LIN {X 0,Y 516.886,Z 290.1,A -85,B 0,C 180,E1 -5001.285,E2 -5001.285} C_VEL
LIN {X 0,Y 516.874,Z 290.104,A -85,B 0,C 180,E1 -5004.22,E2 -5004.22} C_VEL
LIN {X 0,Y 516.884,Z 290.103,A -85,B 0,C 180,E1 -5007.052,E2 -5007.052} C_VEL
LIN {X 0,Y 516.896,Z 290.1,A -85,B 0,C 180,E1 -5009.797,E2 -5009.797} C_VEL
LIN {X 0,Y 516.926,Z 290.096,A -85,B 0,C 180,E1 -5012.467,E2 -5012.467} C_VEL
LIN {X 0,Y 516.86,Z 290.106,A -85,B 0,C 180,E1 -5015.069,E2 -5015.069} C_VEL
LIN {X 0,Y 516.873,Z 290.103,A -85,B 0,C 180,E1 -5017.622,E2 -5017.622} C_VEL
LIN {X 0,Y 516.936,Z 290.095,A -85,B 0,C 180,E1 -5020.13,E2 -5020.13} C_VEL
LIN {X 0,Y 516.909,Z 290.098,A -85,B 0,C 180,E1 -5022.596,E2 -5022.596} C_VEL
LIN {X 0,Y 516.948,Z 290.093,A -85,B 0,C 180,E1 -5025.03,E2 -5025.03} C_VEL
LIN {X 0,Y 516.971,Z 290.091,A -85,B 0,C 180,E1 -5028.234,E2 -5028.234} C_VEL
LIN {X 0,Y 516.96,Z 290.091,A -85,B 0,C 180,E1 -5031.4,E2 -5031.4} C_VEL
LIN {X 0,Y 517.015,Z 290.083,A -85,B 0,C 180,E1 -5033.757,E2 -5033.757} C_VEL
LIN {X 0,Y 517.088,Z 290.074,A -85,B 0,C 180,E1 -5037.663,E2 -5037.663} C_VEL
LIN {X 0,Y 517.097,Z 290.075,A -85,B 0,C 180,E1 -5040.779,E2 -5040.779} C_VEL
LIN {X 0,Y 516.98,Z 290.089,A -85,B 0,C 180,E1 -5043.117,E2 -5043.117} C_VEL
LIN {X 0,Y 516.994,Z 290.088,A -85,B 0,C 180,E1 -5046.243,E2 -5046.243} C_VEL
LIN {X 0,Y 516.948,Z 290.092,A -85,B 0,C 180,E1 -5049.389,E2 -5049.389} C_VEL
LIN {X 0,Y 516.957,Z 290.093,A -85,B 0,C 180,E1 -5051.807,E2 -5051.807} C_VEL
LIN {X 0,Y 516.945,Z 290.093,A -85,B 0,C 180,E1 -5055.144,E2 -5055.144} C_VEL
LIN {X 0,Y 516.918,Z 290.099,A -85,B 0,C 180,E1 -5058.223,E2 -5058.223} C_VEL
LIN {X 0,Y 516.917,Z 290.099,A -85,B 0,C 180,E1 -5060.701,E2 -5060.701} C_VEL
LIN {X 0,Y 516.894,Z 290.099,A -85,B 0,C 180,E1 -5064.073,E2 -5064.073} C_VEL
LIN {X 0,Y 516.895,Z 290.099,A -85,B 0,C 180,E1 -5066.66,E2 -5066.66} C_VEL
LIN {X 0,Y 516.913,Z 290.096,A -85,B 0,C 180,E1 -5069.523,E2 -5069.523} C_VEL
LIN {X 0,Y 516.9,Z 290.102,A -85,B 0,C 180,E1 -5072.543,E2 -5072.543} C_VEL
LIN {X 0,Y 516.867,Z 290.104,A -85,B 0,C 180,E1 -5075.329,E2 -5075.329} C_VEL
LIN {X 0,Y 516.883,Z 290.104,A -85,B 0,C 180,E1 -5077.943,E2 -5077.943} C_VEL
LIN {X 0,Y 516.886,Z 290.101,A -85,B 0,C 180,E1 -5080.742,E2 -5080.742} C_VEL
LIN {X 0,Y 516.885,Z 290.101,A -85,B 0,C 180,E1 -5083.903,E2 -5083.903} C_VEL
LIN {X 0,Y 516.885,Z 290.1,A -85,B 0,C 180,E1 -5086.107,E2 -5086.107} C_VEL
LIN {X 0,Y 516.885,Z 290.1,A -85,B 0,C 180,E1 -5089.258,E2 -5089.258} C_VEL
LIN {X 0,Y 516.916,Z 290.213,A -85,B 0,C 180,E1 -5091.487,E2 -5091.487} C_VEL
LIN {X 0,Y 518.112,Z 296.915,A -85,B 0,C 180,E1 -5093.838,E2 -5093.838} C_VEL
LIN {X 0,Y 518.102,Z 303.042,A -85,B 0,C 180,E1 -5095.839,E2 -5095.839} C_VEL
LIN {X 0,Y 517.763,Z 312.405,A -85,B 0,C 180,E1 -5098.776,E2 -5098.776} C_VEL
LIN {X 0,Y 517.485,Z 322.995,A -85,B 0,C 180,E1 -5101.979,E2 -5101.979} C_VEL
LIN {X 0,Y 517.191,Z 333.621,A -85,B 0,C 180,E1 -5105.086,E2 -5105.086} C_VEL
LIN {X 0,Y 516.956,Z 344.077,A -85,B 0,C 180,E1 -5108.046,E2 -5108.046} C_VEL
LIN {X 0,Y 516.804,Z 354.493,A -85,B 0,C 180,E1 -5110.951,E2 -5110.951} C_VEL
LIN {X 0,Y 516.651,Z 364.97,A -85,B 0,C 180,E1 -5113.808,E2 -5113.808} C_VEL
LIN {X 0,Y 516.565,Z 373.407,A -85,B 0,C 180,E1 -5116.075,E2 -5116.075} C_VEL
LIN {X 0,Y 518.411,Z 387.284,A -85,B 0,C 180,E1 -5116.451,E2 -5116.451} C_VEL
LIN {X 0,Y 518.142,Z 400.417,A -85,B 0,C 180,E1 -5116.918,E2 -5116.918} C_VEL
LIN {X 0,Y 517.84,Z 412.913,A -85,B 0,C 180,E1 -5117.534,E2 -5117.534} C_VEL
LIN {X 0,Y 517.512,Z 424.089,A -85,B 0,C 180,E1 -5118.246,E2 -5118.246} C_VEL
LIN {X 0,Y 517.241,Z 435.096,A -85,B 0,C 180,E1 -5119.133,E2 -5119.133} C_VEL
LIN {X 0,Y 516.978,Z 444.068,A -85,B 0,C 180,E1 -5120.019,E2 -5120.019} C_VEL
LIN {X 0,Y 516.739,Z 453.823,A -85,B 0,C 180,E1 -5121.199,E2 -5121.199} C_VEL
LIN {X 0,Y 516.556,Z 461.599,A -85,B 0,C 180,E1 -5122.377,E2 -5122.377} C_VEL
LIN {X 0,Y 516.412,Z 468.766,A -85,B 0,C 180,E1 -5123.75,E2 -5123.75} C_VEL
LIN {X 0,Y 516.313,Z 473.535,A -85,B 0,C 180,E1 -5124.924,E2 -5124.924} C_VEL
LIN {X 0,Y 516.37,Z 477.189,A -85,B 0,C 180,E1 -5126.098,E2 -5126.098} C_VEL
LIN {X 0,Y 516.282,Z 479.064,A -85,B 0,C 180,E1 -5126.879,E2 -5126.879} C_VEL
LIN {X 0,Y 516.261,Z 480.474,A -85,B 0,C 180,E1 -5127.659,E2 -5127.659} C_VEL
LIN {X 0,Y 516.169,Z 482.086,A -85,B 0,C 180,E1 -5129.22,E2 -5129.22} C_VEL
LIN {X 0,Y 516.167,Z 482.301,A -85,B 0,C 180,E1 -5130,E2 -5130} C_VEL
LIN {X 0,Y 516.17,Z 482.08,A -85,B 0,C 180,E1 -5130.78,E2 -5130.78} C_VEL
LIN {X 0,Y 516.261,Z 480.461,A -85,B 0,C 180,E1 -5132.341,E2 -5132.341} C_VEL
LIN {X 0,Y 516.296,Z 479.044,A -85,B 0,C 180,E1 -5133.121,E2 -5133.121} C_VEL
LIN {X 0,Y 516.331,Z 476.068,A -85,B 0,C 180,E1 -5134.293,E2 -5134.293} C_VEL
LIN {X 0,Y 516.402,Z 472.041,A -85,B 0,C 180,E1 -5135.467,E2 -5135.467} C_VEL
LIN {X 0,Y 516.456,Z 466.027,A -85,B 0,C 180,E1 -5136.804,E2 -5136.804} C_VEL
LIN {X 0,Y 516.605,Z 459.082,A -85,B 0,C 180,E1 -5138.016,E2 -5138.016} C_VEL
LIN {X 0,Y 516.803,Z 450.691,A -85,B 0,C 180,E1 -5139.195,E2 -5139.195} C_VEL
LIN {X 0,Y 517.03,Z 442.093,A -85,B 0,C 180,E1 -5140.178,E2 -5140.178} C_VEL
LIN {X 0,Y 517.361,Z 431.487,A -85,B 0,C 180,E1 -5141.162,E2 -5141.162} C_VEL
LIN {X 0,Y 517.599,Z 420.41,A -85,B 0,C 180,E1 -5141.991,E2 -5141.991} C_VEL
LIN {X 0,Y 517.909,Z 409.518,A -85,B 0,C 180,E1 -5142.64,E2 -5142.64} C_VEL
LIN {X 0,Y 518.191,Z 397.722,A -85,B 0,C 180,E1 -5143.181,E2 -5143.181} C_VEL
LIN {X 0,Y 518.32,Z 385.546,A -85,B 0,C 180,E1 -5143.589,E2 -5143.589} C_VEL
LIN {X 0,Y 516.564,Z 373.094,A -85,B 0,C 180,E1 -5143.925,E2 -5143.925} C_VEL
LIN {X 0,Y 516.683,Z 361.513,A -85,B 0,C 180,E1 -5147.005,E2 -5147.005} C_VEL
LIN {X 0,Y 516.8,Z 350.765,A -85,B 0,C 180,E1 -5149.876,E2 -5149.876} C_VEL
LIN {X 0,Y 516.945,Z 340.244,A -85,B 0,C 180,E1 -5152.797,E2 -5152.797} C_VEL
LIN {X 0,Y 517.154,Z 329.607,A -85,B 0,C 180,E1 -5155.777,E2 -5155.777} C_VEL
LIN {X 0,Y 517.35,Z 319.161,A -85,B 0,C 180,E1 -5158.833,E2 -5158.833} C_VEL
LIN {X 0,Y 517.601,Z 310.272,A -85,B 0,C 180,E1 -5161.537,E2 -5161.537} C_VEL
LIN {X 0,Y 517.915,Z 302.102,A -85,B 0,C 180,E1 -5164.131,E2 -5164.131} C_VEL
LIN {X 0,Y 518.09,Z 297.453,A -85,B 0,C 180,E1 -5165.684,E2 -5165.684} C_VEL
LIN {X 0,Y 517.081,Z 291.154,A -85,B 0,C 180,E1 -5167.971,E2 -5167.971} C_VEL
LIN {X 0,Y 516.893,Z 290.102,A -85,B 0,C 180,E1 -5168.408,E2 -5168.408} C_VEL
LIN {X 0,Y 516.916,Z 290.099,A -85,B 0,C 180,E1 -5171.775,E2 -5171.775} C_VEL
LIN {X 0,Y 516.927,Z 290.1,A -85,B 0,C 180,E1 -5175.01,E2 -5175.01} C_VEL
LIN {X 0,Y 516.918,Z 290.099,A -85,B 0,C 180,E1 -5178.399,E2 -5178.399} C_VEL
LIN {X 0,Y 516.888,Z 290.103,A -85,B 0,C 180,E1 -5181.284,E2 -5181.284} C_VEL
LIN {X 0,Y 516.876,Z 290.104,A -85,B 0,C 180,E1 -5184.22,E2 -5184.22} C_VEL
LIN {X 0,Y 516.9,Z 290.102,A -85,B 0,C 180,E1 -5187.053,E2 -5187.053} C_VEL
LIN {X 0,Y 516.898,Z 290.1,A -85,B 0,C 180,E1 -5189.796,E2 -5189.796} C_VEL
LIN {X 0,Y 516.934,Z 290.095,A -85,B 0,C 180,E1 -5192.468,E2 -5192.468} C_VEL
LIN {X 0,Y 516.915,Z 290.099,A -85,B 0,C 180,E1 -5195.072,E2 -5195.072} C_VEL
LIN {X 0,Y 516.891,Z 290.101,A -85,B 0,C 180,E1 -5198.462,E2 -5198.462} C_VEL
LIN {X 0,Y 516.906,Z 290.1,A -85,B 0,C 180,E1 -5200.955,E2 -5200.955} C_VEL
LIN {X 0,Y 516.913,Z 290.098,A -85,B 0,C 180,E1 -5203.41,E2 -5203.41} C_VEL
LIN {X 0,Y 516.901,Z 290.1,A -85,B 0,C 180,E1 -5205.834,E2 -5205.834} C_VEL
LIN {X 0,Y 516.972,Z 290.092,A -85,B 0,C 180,E1 -5208.234,E2 -5208.234} C_VEL
LIN {X 0,Y 516.961,Z 290.092,A -85,B 0,C 180,E1 -5211.399,E2 -5211.399} C_VEL
LIN {X 0,Y 517.028,Z 290.084,A -85,B 0,C 180,E1 -5214.54,E2 -5214.54} C_VEL
LIN {X 0,Y 517.09,Z 290.076,A -85,B 0,C 180,E1 -5217.663,E2 -5217.663} C_VEL
LIN {X 0,Y 517.098,Z 290.075,A -85,B 0,C 180,E1 -5220.779,E2 -5220.779} C_VEL
LIN {X 0,Y 517.018,Z 290.087,A -85,B 0,C 180,E1 -5223.117,E2 -5223.117} C_VEL
LIN {X 0,Y 516.995,Z 290.09,A -85,B 0,C 180,E1 -5226.243,E2 -5226.243} C_VEL
LIN {X 0,Y 516.922,Z 290.098,A -85,B 0,C 180,E1 -5228.601,E2 -5228.601} C_VEL
LIN {X 0,Y 516.657,Z 290.133,A -85,B 0,C 180,E1 -5231.773,E2 -5231.773} C_VEL
LIN {X 0,Y 516.591,Z 293.302,A -85,B 0,C 180,E1 -5234.999,E2 -5234.999} C_VEL
LIN {X 0,Y 516.441,Z 296.476,A -85,B 0,C 180,E1 -5238.24,E2 -5238.24} C_VEL
LIN {X 0,Y 516.408,Z 298.931,A -85,B 0,C 180,E1 -5240.723,E2 -5240.723} C_VEL
LIN {X 0,Y 516.353,Z 301.393,A -85,B 0,C 180,E1 -5243.248,E2 -5243.248} C_VEL
LIN {X 0,Y 516.359,Z 302.348,A -85,B 0,C 180,E1 -5244.201,E2 -5244.201} C_VEL
LIN {X 0,Y 518.52,Z 312.656,A -85,B 0,C 180,E1 -5244.55,E2 -5244.55} C_VEL
LIN {X 0,Y 518.316,Z 325.138,A -85,B 0,C 180,E1 -5245.017,E2 -5245.017} C_VEL
LIN {X 0,Y 518.014,Z 337.109,A -85,B 0,C 180,E1 -5245.623,E2 -5245.623} C_VEL
LIN {X 0,Y 517.73,Z 348.451,A -85,B 0,C 180,E1 -5246.371,E2 -5246.371} C_VEL
LIN {X 0,Y 517.383,Z 359.408,A -85,B 0,C 180,E1 -5247.287,E2 -5247.287} C_VEL
LIN {X 0,Y 517.126,Z 368.926,A -85,B 0,C 180,E1 -5248.274,E2 -5248.274} C_VEL
LIN {X 0,Y 516.91,Z 377.037,A -85,B 0,C 180,E1 -5249.305,E2 -5249.305} C_VEL
LIN {X 0,Y 516.702,Z 384.138,A -85,B 0,C 180,E1 -5250.413,E2 -5250.413} C_VEL
LIN {X 0,Y 516.554,Z 390.225,A -85,B 0,C 180,E1 -5251.588,E2 -5251.588} C_VEL
LIN {X 0,Y 516.396,Z 395.846,A -85,B 0,C 180,E1 -5252.983,E2 -5252.983} C_VEL
LIN {X 0,Y 516.307,Z 399.976,A -85,B 0,C 180,E1 -5254.395,E2 -5254.395} C_VEL
LIN {X 0,Y 516.235,Z 402.698,A -85,B 0,C 180,E1 -5255.831,E2 -5255.831} C_VEL
LIN {X 0,Y 516.188,Z 403.797,A -85,B 0,C 180,E1 -5256.803,E2 -5256.803} C_VEL
LIN {X 0,Y 516.184,Z 404.25,A -85,B 0,C 180,E1 -5257.843,E2 -5257.843} C_VEL
LIN {X 0,Y 516.212,Z 403.894,A -85,B 0,C 180,E1 -5259.101,E2 -5259.101} C_VEL
LIN {X 0,Y 516.221,Z 402.572,A -85,B 0,C 180,E1 -5260.323,E2 -5260.323} C_VEL
LIN {X 0,Y 516.346,Z 399.485,A -85,B 0,C 180,E1 -5261.866,E2 -5261.866} C_VEL
LIN {X 0,Y 516.451,Z 394.859,A -85,B 0,C 180,E1 -5263.358,E2 -5263.358} C_VEL
LIN {X 0,Y 516.535,Z 389.155,A -85,B 0,C 180,E1 -5264.71,E2 -5264.71} C_VEL
LIN {X 0,Y 516.554,Z 387.672,A -85,B 0,C 180,E1 -5265.004,E2 -5265.004} C_VEL
LIN {X 0,Y 515.988,Z 384.738,A -85,B 0,C 180,E1 -5265.569,E2 -5265.569} C_VEL
LIN {X 0,Y 513.309,Z 379.676,A -85,B 0,C 180,E1 -5266.469,E2 -5266.469} C_VEL
LIN {X 0,Y 510.647,Z 374.075,A -85,B 0,C 180,E1 -5267.333,E2 -5267.333} C_VEL
LIN {X 0,Y 510.116,Z 370.186,A -85,B 0,C 180,E1 -5267.836,E2 -5267.836} C_VEL
LIN {X 0,Y 510.386,Z 361.354,A -85,B 0,C 180,E1 -5268.791,E2 -5268.791} C_VEL
LIN {X 0,Y 510.668,Z 351.025,A -85,B 0,C 180,E1 -5269.696,E2 -5269.696} C_VEL
LIN {X 0,Y 510.966,Z 340.365,A -85,B 0,C 180,E1 -5270.449,E2 -5270.449} C_VEL
LIN {X 0,Y 511.327,Z 328.624,A -85,B 0,C 180,E1 -5271.1,E2 -5271.1} C_VEL
LIN {X 0,Y 511.56,Z 316.145,A -85,B 0,C 180,E1 -5271.614,E2 -5271.614} C_VEL
LIN {X 0,Y 511.334,Z 312.242,A -85,B 0,C 180,E1 -5271.752,E2 -5271.752} C_VEL
LIN {X 0,Y 509.237,Z 302.327,A -85,B 0,C 180,E1 -5272.084,E2 -5272.084} C_VEL
LIN {X 0,Y 509.256,Z 299.712,A -85,B 0,C 180,E1 -5274.576,E2 -5274.576} C_VEL
LIN {X 0,Y 509.286,Z 296.717,A -85,B 0,C 180,E1 -5277.439,E2 -5277.439} C_VEL
LIN {X 0,Y 509.35,Z 293.644,A -85,B 0,C 180,E1 -5280.374,E2 -5280.374} C_VEL
LIN {X 0,Y 509.375,Z 291.039,A -85,B 0,C 180,E1 -5282.915,E2 -5282.915} C_VEL
LIN {X 0,Y 509.662,Z 291.003,A -85,B 0,C 180,E1 -5285.563,E2 -5285.563} C_VEL
LIN {X 0,Y 509.823,Z 290.981,A -85,B 0,C 180,E1 -5288.148,E2 -5288.148} C_VEL
LIN {X 0,Y 509.859,Z 290.976,A -85,B 0,C 180,E1 -5290.681,E2 -5290.681} C_VEL
LIN {X 0,Y 509.872,Z 290.975,A -85,B 0,C 180,E1 -5293.174,E2 -5293.174} C_VEL
LIN {X 0,Y 509.863,Z 290.975,A -85,B 0,C 180,E1 -5295.634,E2 -5295.634} C_VEL
LIN {X 0,Y 509.914,Z 290.971,A -85,B 0,C 180,E1 -5298.874,E2 -5298.874} C_VEL
LIN {X 0,Y 509.953,Z 290.962,A -85,B 0,C 180,E1 -5302.078,E2 -5302.078} C_VEL
LIN {X 0,Y 509.974,Z 290.962,A -85,B 0,C 180,E1 -5304.464,E2 -5304.464} C_VEL
LIN {X 0,Y 510.056,Z 290.952,A -85,B 0,C 180,E1 -5307.631,E2 -5307.631} C_VEL
LIN {X 0,Y 510.064,Z 290.951,A -85,B 0,C 180,E1 -5310.789,E2 -5310.789} C_VEL
LIN {X 0,Y 509.957,Z 290.965,A -85,B 0,C 180,E1 -5313.16,E2 -5313.16} C_VEL
LIN {X 0,Y 509.936,Z 290.966,A -85,B 0,C 180,E1 -5316.33,E2 -5316.33} C_VEL
LIN {X 0,Y 509.912,Z 290.97,A -85,B 0,C 180,E1 -5318.72,E2 -5318.72} C_VEL
LIN {X 0,Y 509.906,Z 290.969,A -85,B 0,C 180,E1 -5321.932,E2 -5321.932} C_VEL
LIN {X 0,Y 509.896,Z 290.971,A -85,B 0,C 180,E1 -5325.242,E2 -5325.242} C_VEL
LIN {X 0,Y 509.858,Z 290.976,A -85,B 0,C 180,E1 -5328.484,E2 -5328.484} C_VEL
LIN {X 0,Y 509.852,Z 290.976,A -85,B 0,C 180,E1 -5331.002,E2 -5331.002} C_VEL
LIN {X 0,Y 509.872,Z 290.975,A -85,B 0,C 180,E1 -5334.426,E2 -5334.426} C_VEL
LIN {X 0,Y 509.884,Z 290.973,A -85,B 0,C 180,E1 -5337.056,E2 -5337.056} C_VEL
LIN {X 0,Y 509.858,Z 290.977,A -85,B 0,C 180,E1 -5339.751,E2 -5339.751} C_VEL
LIN {X 0,Y 509.869,Z 290.974,A -85,B 0,C 180,E1 -5342.773,E2 -5342.773} C_VEL
LIN {X 0,Y 509.827,Z 290.979,A -85,B 0,C 180,E1 -5345.579,E2 -5345.579} C_VEL
LIN {X 0,Y 509.852,Z 290.978,A -85,B 0,C 180,E1 -5348.338,E2 -5348.338} C_VEL
LIN {X 0,Y 509.858,Z 290.978,A -85,B 0,C 180,E1 -5351.426,E2 -5351.426} C_VEL
LIN {X 0,Y 509.841,Z 290.977,A -85,B 0,C 180,E1 -5354.67,E2 -5354.67} C_VEL
LIN {X 0,Y 509.86,Z 290.976,A -85,B 0,C 180,E1 -5358.103,E2 -5358.103} C_VEL
LIN {X 0,Y 509.851,Z 290.977,A -85,B 0,C 180,E1 -5360.648,E2 -5360.648} C_VEL
LIN {X 0,Y 509.828,Z 290.98,A -85,B 0,C 180,E1 -5363.647,E2 -5363.647} C_VEL
LIN {X 0,Y 509.845,Z 290.977,A -85,B 0,C 180,E1 -5366.538,E2 -5366.538} C_VEL
LIN {X 0,Y 509.849,Z 290.978,A -85,B 0,C 180,E1 -5369.335,E2 -5369.335} C_VEL
LIN {X 0,Y 509.888,Z 290.974,A -85,B 0,C 180,E1 -5372.054,E2 -5372.054} C_VEL
LIN {X 0,Y 509.82,Z 290.981,A -85,B 0,C 180,E1 -5374.701,E2 -5374.701} C_VEL
LIN {X 0,Y 509.83,Z 290.982,A -85,B 0,C 180,E1 -5377.458,E2 -5377.458} C_VEL
LIN {X 0,Y 509.921,Z 290.969,A -85,B 0,C 180,E1 -5379.845,E2 -5379.845} C_VEL
LIN {X 0,Y 509.873,Z 290.974,A -85,B 0,C 180,E1 -5383.174,E2 -5383.174} C_VEL
LIN {X 0,Y 509.867,Z 290.975,A -85,B 0,C 180,E1 -5385.634,E2 -5385.634} C_VEL
LIN {X 0,Y 509.919,Z 290.968,A -85,B 0,C 180,E1 -5388.875,E2 -5388.875} C_VEL
LIN {X 0,Y 509.926,Z 290.968,A -85,B 0,C 180,E1 -5392.078,E2 -5392.078} C_VEL
LIN {X 0,Y 509.984,Z 290.961,A -85,B 0,C 180,E1 -5394.464,E2 -5394.464} C_VEL
LIN {X 0,Y 510.058,Z 290.95,A -85,B 0,C 180,E1 -5397.631,E2 -5397.631} C_VEL
LIN {X 0,Y 510.068,Z 290.95,A -85,B 0,C 180,E1 -5400.79,E2 -5400.79} C_VEL
LIN {X 0,Y 509.923,Z 290.968,A -85,B 0,C 180,E1 -5403.16,E2 -5403.16} C_VEL
LIN {X 0,Y 509.94,Z 290.967,A -85,B 0,C 180,E1 -5406.33,E2 -5406.33} C_VEL
LIN {X 0,Y 509.888,Z 290.97,A -85,B 0,C 180,E1 -5409.521,E2 -5409.521} C_VEL
LIN {X 0,Y 509.91,Z 290.97,A -85,B 0,C 180,E1 -5411.932,E2 -5411.932} C_VEL
LIN {X 0,Y 509.9,Z 290.972,A -85,B 0,C 180,E1 -5415.242,E2 -5415.242} C_VEL
LIN {X 0,Y 509.862,Z 290.976,A -85,B 0,C 180,E1 -5418.484,E2 -5418.484} C_VEL
LIN {X 0,Y 509.855,Z 290.976,A -85,B 0,C 180,E1 -5421.002,E2 -5421.002} C_VEL
LIN {X 0,Y 509.826,Z 290.981,A -85,B 0,C 180,E1 -5423.564,E2 -5423.564} C_VEL
LIN {X 0,Y 509.88,Z 290.974,A -85,B 0,C 180,E1 -5426.37,E2 -5426.37} C_VEL
LIN {X 0,Y 509.863,Z 290.975,A -85,B 0,C 180,E1 -5429.726,E2 -5429.726} C_VEL
LIN {X 0,Y 509.878,Z 290.974,A -85,B 0,C 180,E1 -5432.774,E2 -5432.774} C_VEL
LIN {X 0,Y 509.827,Z 290.981,A -85,B 0,C 180,E1 -5435.578,E2 -5435.578} C_VEL
LIN {X 0,Y 509.853,Z 290.976,A -85,B 0,C 180,E1 -5438.338,E2 -5438.338} C_VEL
LIN {X 0,Y 509.856,Z 290.975,A -85,B 0,C 180,E1 -5441.426,E2 -5441.426} C_VEL
LIN {X 0,Y 509.843,Z 290.978,A -85,B 0,C 180,E1 -5444.67,E2 -5444.67} C_VEL
LIN {X 0,Y 509.853,Z 290.977,A -85,B 0,C 180,E1 -5448.104,E2 -5448.104} C_VEL
LIN {X 0,Y 509.87,Z 291.038,A -85,B 0,C 180,E1 -5451.222,E2 -5451.222} C_VEL
LIN {X 0,Y 511.143,Z 298.136,A -85,B 0,C 180,E1 -5453.755,E2 -5453.755} C_VEL
LIN {X 0,Y 511.132,Z 303.947,A -85,B 0,C 180,E1 -5455.684,E2 -5455.684} C_VEL
LIN {X 0,Y 510.801,Z 312.904,A -85,B 0,C 180,E1 -5458.545,E2 -5458.545} C_VEL
LIN {X 0,Y 510.463,Z 323.424,A -85,B 0,C 180,E1 -5461.781,E2 -5461.781} C_VEL
LIN {X 0,Y 510.136,Z 334.637,A -85,B 0,C 180,E1 -5465.11,E2 -5465.11} C_VEL
LIN {X 0,Y 509.878,Z 345.171,A -85,B 0,C 180,E1 -5468.151,E2 -5468.151} C_VEL
LIN {X 0,Y 509.726,Z 355.603,A -85,B 0,C 180,E1 -5471.094,E2 -5471.094} C_VEL
LIN {X 0,Y 509.572,Z 366.002,A -85,B 0,C 180,E1 -5473.988,E2 -5473.988} C_VEL
LIN {X 0,Y 509.485,Z 372.903,A -85,B 0,C 180,E1 -5475.878,E2 -5475.878} C_VEL
LIN {X 0,Y 511.45,Z 388.36,A -85,B 0,C 180,E1 -5476.313,E2 -5476.313} C_VEL
LIN {X 0,Y 511.183,Z 400.988,A -85,B 0,C 180,E1 -5476.787,E2 -5476.787} C_VEL
LIN {X 0,Y 510.815,Z 414.088,A -85,B 0,C 180,E1 -5477.46,E2 -5477.46} C_VEL
LIN {X 0,Y 510.423,Z 426.17,A -85,B 0,C 180,E1 -5478.282,E2 -5478.282} C_VEL
LIN {X 0,Y 510.199,Z 436.704,A -85,B 0,C 180,E1 -5479.182,E2 -5479.182} C_VEL
LIN {X 0,Y 509.878,Z 445.319,A -85,B 0,C 180,E1 -5480.079,E2 -5480.079} C_VEL
LIN {X 0,Y 509.689,Z 453.281,A -85,B 0,C 180,E1 -5481.076,E2 -5481.076} C_VEL
LIN {X 0,Y 509.483,Z 461.063,A -85,B 0,C 180,E1 -5482.271,E2 -5482.271} C_VEL
LIN {X 0,Y 509.322,Z 467.345,A -85,B 0,C 180,E1 -5483.47,E2 -5483.47} C_VEL
LIN {X 0,Y 509.247,Z 473.005,A -85,B 0,C 180,E1 -5484.853,E2 -5484.853} C_VEL
LIN {X 0,Y 509.296,Z 476.66,A -85,B 0,C 180,E1 -5486.044,E2 -5486.044} C_VEL
LIN {X 0,Y 509.201,Z 478.534,A -85,B 0,C 180,E1 -5486.835,E2 -5486.835} C_VEL
LIN {X 0,Y 509.19,Z 479.945,A -85,B 0,C 180,E1 -5487.627,E2 -5487.627} C_VEL
LIN {X 0,Y 509.089,Z 481.554,A -85,B 0,C 180,E1 -5489.209,E2 -5489.209} C_VEL
LIN {X 0,Y 509.088,Z 481.767,A -85,B 0,C 180,E1 -5490,E2 -5490} C_VEL
LIN {X 0,Y 509.09,Z 481.544,A -85,B 0,C 180,E1 -5490.791,E2 -5490.791} C_VEL
LIN {X 0,Y 509.191,Z 479.917,A -85,B 0,C 180,E1 -5492.373,E2 -5492.373} C_VEL
LIN {X 0,Y 509.214,Z 478.495,A -85,B 0,C 180,E1 -5493.165,E2 -5493.165} C_VEL
LIN {X 0,Y 509.242,Z 475.511,A -85,B 0,C 180,E1 -5494.353,E2 -5494.353} C_VEL
LIN {X 0,Y 509.338,Z 471.477,A -85,B 0,C 180,E1 -5495.543,E2 -5495.543} C_VEL
LIN {X 0,Y 509.392,Z 465.727,A -85,B 0,C 180,E1 -5496.845,E2 -5496.845} C_VEL
LIN {X 0,Y 509.527,Z 458.492,A -85,B 0,C 180,E1 -5498.128,E2 -5498.128} C_VEL
LIN {X 0,Y 509.754,Z 450.088,A -85,B 0,C 180,E1 -5499.323,E2 -5499.323} C_VEL
LIN {X 0,Y 509.992,Z 441.475,A -85,B 0,C 180,E1 -5500.32,E2 -5500.32} C_VEL
LIN {X 0,Y 510.325,Z 430.854,A -85,B 0,C 180,E1 -5501.318,E2 -5501.318} C_VEL
LIN {X 0,Y 510.587,Z 419.764,A -85,B 0,C 180,E1 -5502.158,E2 -5502.158} C_VEL
LIN {X 0,Y 510.954,Z 408.862,A -85,B 0,C 180,E1 -5502.815,E2 -5502.815} C_VEL
LIN {X 0,Y 511.237,Z 397.043,A -85,B 0,C 180,E1 -5503.363,E2 -5503.363} C_VEL
LIN {X 0,Y 511.308,Z 386.224,A -85,B 0,C 180,E1 -5503.741,E2 -5503.741} C_VEL
LIN {X 0,Y 509.571,Z 373.669,A -85,B 0,C 180,E1 -5504.081,E2 -5504.081} C_VEL
LIN {X 0,Y 509.478,Z 372.485,A -85,B 0,C 180,E1 -5504.122,E2 -5504.122} C_VEL
LIN {X 0,Y 509.628,Z 360.94,A -85,B 0,C 180,E1 -5507.247,E2 -5507.247} C_VEL
LIN {X 0,Y 509.784,Z 349.53,A -85,B 0,C 180,E1 -5510.37,E2 -5510.37} C_VEL
LIN {X 0,Y 509.929,Z 338.207,A -85,B 0,C 180,E1 -5513.559,E2 -5513.559} C_VEL
LIN {X 0,Y 510.16,Z 327.415,A -85,B 0,C 180,E1 -5516.691,E2 -5516.691} C_VEL
LIN {X 0,Y 510.442,Z 316.906,A -85,B 0,C 180,E1 -5519.84,E2 -5519.84} C_VEL
LIN {X 0,Y 510.802,Z 307.112,A -85,B 0,C 180,E1 -5522.935,E2 -5522.935} C_VEL
LIN {X 0,Y 511.128,Z 298.601,A -85,B 0,C 180,E1 -5525.782,E2 -5525.782} C_VEL
LIN {X 0,Y 510.038,Z 291.998,A -85,B 0,C 180,E1 -5528.24,E2 -5528.24} C_VEL
LIN {X 0,Y 509.879,Z 290.974,A -85,B 0,C 180,E1 -5528.714,E2 -5528.714} C_VEL
LIN {X 0,Y 509.86,Z 290.978,A -85,B 0,C 180,E1 -5531.897,E2 -5531.897} C_VEL
LIN {X 0,Y 509.861,Z 290.98,A -85,B 0,C 180,E1 -5535.332,E2 -5535.332} C_VEL
LIN {X 0,Y 509.86,Z 290.978,A -85,B 0,C 180,E1 -5538.575,E2 -5538.575} C_VEL
LIN {X 0,Y 509.856,Z 290.978,A -85,B 0,C 180,E1 -5541.786,E2 -5541.786} C_VEL
LIN {X 0,Y 509.835,Z 290.98,A -85,B 0,C 180,E1 -5544.622,E2 -5544.622} C_VEL
LIN {X 0,Y 509.866,Z 290.976,A -85,B 0,C 180,E1 -5547.481,E2 -5547.481} C_VEL
LIN {X 0,Y 509.864,Z 290.977,A -85,B 0,C 180,E1 -5550.274,E2 -5550.274} C_VEL
LIN {X 0,Y 509.891,Z 290.974,A -85,B 0,C 180,E1 -5552.945,E2 -5552.945} C_VEL
LIN {X 0,Y 509.87,Z 290.973,A -85,B 0,C 180,E1 -5555.574,E2 -5555.574} C_VEL
LIN {X 0,Y 509.856,Z 290.979,A -85,B 0,C 180,E1 -5558.998,E2 -5558.998} C_VEL
LIN {X 0,Y 509.867,Z 290.975,A -85,B 0,C 180,E1 -5561.516,E2 -5561.516} C_VEL
LIN {X 0,Y 509.917,Z 290.969,A -85,B 0,C 180,E1 -5564.819,E2 -5564.819} C_VEL
LIN {X 0,Y 509.907,Z 290.972,A -85,B 0,C 180,E1 -5568.124,E2 -5568.124} C_VEL
LIN {X 0,Y 509.91,Z 290.971,A -85,B 0,C 180,E1 -5571.28,E2 -5571.28} C_VEL
LIN {X 0,Y 509.979,Z 290.962,A -85,B 0,C 180,E1 -5574.464,E2 -5574.464} C_VEL
LIN {X 0,Y 510.061,Z 290.951,A -85,B 0,C 180,E1 -5577.631,E2 -5577.631} C_VEL
LIN {X 0,Y 510.069,Z 290.95,A -85,B 0,C 180,E1 -5580.789,E2 -5580.789} C_VEL
LIN {X 0,Y 509.96,Z 290.966,A -85,B 0,C 180,E1 -5583.16,E2 -5583.16} C_VEL
LIN {X 0,Y 509.943,Z 290.967,A -85,B 0,C 180,E1 -5586.33,E2 -5586.33} C_VEL
LIN {X 0,Y 509.864,Z 290.977,A -85,B 0,C 180,E1 -5588.721,E2 -5588.721} C_VEL
LIN {X 0,Y 509.589,Z 291.091,A -85,B 0,C 180,E1 -5591.939,E2 -5591.939} C_VEL
LIN {X 0,Y 509.529,Z 294.259,A -85,B 0,C 180,E1 -5595.193,E2 -5595.193} C_VEL
LIN {X 0,Y 509.389,Z 297.53,A -85,B 0,C 180,E1 -5598.501,E2 -5598.501} C_VEL
LIN {X 0,Y 509.343,Z 300.019,A -85,B 0,C 180,E1 -5601.024,E2 -5601.024} C_VEL
LIN {X 0,Y 509.32,Z 302.967,A -85,B 0,C 180,E1 -5604.02,E2 -5604.02} C_VEL
LIN {X 0,Y 511.581,Z 313.227,A -85,B 0,C 180,E1 -5604.366,E2 -5604.366} C_VEL
LIN {X 0,Y 511.41,Z 325.963,A -85,B 0,C 180,E1 -5604.853,E2 -5604.853} C_VEL
LIN {X 0,Y 511.114,Z 337.529,A -85,B 0,C 180,E1 -5605.448,E2 -5605.448} C_VEL
LIN {X 0,Y 510.81,Z 347.766,A -85,B 0,C 180,E1 -5606.121,E2 -5606.121} C_VEL
LIN {X 0,Y 510.494,Z 358.668,A -85,B 0,C 180,E1 -5607.021,E2 -5607.021} C_VEL
LIN {X 0,Y 510.193,Z 367.589,A -85,B 0,C 180,E1 -5607.928,E2 -5607.928} C_VEL
LIN {X 0,Y 509.958,Z 376.696,A -85,B 0,C 180,E1 -5609.065,E2 -5609.065} C_VEL
LIN {X 0,Y 509.702,Z 384.172,A -85,B 0,C 180,E1 -5610.217,E2 -5610.217} C_VEL
LIN {X 0,Y 509.501,Z 391.273,A -85,B 0,C 180,E1 -5611.612,E2 -5611.612} C_VEL
LIN {X 0,Y 509.341,Z 396.89,A -85,B 0,C 180,E1 -5613.058,E2 -5613.058} C_VEL
LIN {X 0,Y 509.237,Z 400.775,A -85,B 0,C 180,E1 -5614.461,E2 -5614.461} C_VEL
LIN {X 0,Y 509.164,Z 402.768,A -85,B 0,C 180,E1 -5615.473,E2 -5615.473} C_VEL
LIN {X 0,Y 509.121,Z 404.35,A -85,B 0,C 180,E1 -5616.808,E2 -5616.808} C_VEL
LIN {X 0,Y 509.098,Z 404.812,A -85,B 0,C 180,E1 -5618.105,E2 -5618.105} C_VEL
LIN {X 0,Y 509.15,Z 404.202,A -85,B 0,C 180,E1 -5619.417,E2 -5619.417} C_VEL
LIN {X 0,Y 509.158,Z 402.726,A -85,B 0,C 180,E1 -5620.608,E2 -5620.608} C_VEL
LIN {X 0,Y 509.297,Z 400.243,A -85,B 0,C 180,E1 -5621.826,E2 -5621.826} C_VEL
LIN {X 0,Y 509.394,Z 395.914,A -85,B 0,C 180,E1 -5623.279,E2 -5623.279} C_VEL
LIN {X 0,Y 509.503,Z 390.094,A -85,B 0,C 180,E1 -5624.707,E2 -5624.707} C_VEL
LIN {X 0,Y 509.64,Z 384.324,A -85,B 0,C 180,E1 -5625.814,E2 -5625.814} C_VEL
LIN {X 0,Y 509.875,Z 377.18,A -85,B 0,C 180,E1 -5626.932,E2 -5626.932} C_VEL
LIN {X 0,Y 510.116,Z 370.186,A -85,B 0,C 180,E1 -5627.836,E2 -5627.836} C_VEL
LIN {X 0,Y 509.595,Z 366.184,A -85,B 0,C 180,E1 -5628.322,E2 -5628.322} C_VEL
LIN {X 0,Y 507,Z 359.435,A -85,B 0,C 180,E1 -5629.089,E2 -5629.089} C_VEL
LIN {X 0,Y 504.409,Z 352.16,A -85,B 0,C 180,E1 -5629.793,E2 -5629.793} C_VEL
LIN {X 0,Y 503.89,Z 347.336,A -85,B 0,C 180,E1 -5630.175,E2 -5630.175} C_VEL
LIN {X 0,Y 504.231,Z 336.228,A -85,B 0,C 180,E1 -5630.898,E2 -5630.898} C_VEL
LIN {X 0,Y 504.576,Z 323.811,A -85,B 0,C 180,E1 -5631.521,E2 -5631.521} C_VEL
LIN {X 0,Y 504.532,Z 313.781,A -85,B 0,C 180,E1 -5631.902,E2 -5631.902} C_VEL
LIN {X 0,Y 502.159,Z 302.799,A -85,B 0,C 180,E1 -5632.285,E2 -5632.285} C_VEL
LIN {X 0,Y 502.183,Z 299.952,A -85,B 0,C 180,E1 -5634.985,E2 -5634.985} C_VEL
LIN {X 0,Y 502.21,Z 296.941,A -85,B 0,C 180,E1 -5637.874,E2 -5637.874} C_VEL
LIN {X 0,Y 502.265,Z 293.995,A -85,B 0,C 180,E1 -5640.676,E2 -5640.676} C_VEL
LIN {X 0,Y 502.282,Z 292.089,A -85,B 0,C 180,E1 -5642.5,E2 -5642.5} C_VEL
LIN {X 0,Y 502.593,Z 291.884,A -85,B 0,C 180,E1 -5645.357,E2 -5645.357} C_VEL
LIN {X 0,Y 502.769,Z 291.859,A -85,B 0,C 180,E1 -5647.826,E2 -5647.826} C_VEL
LIN {X 0,Y 502.822,Z 291.851,A -85,B 0,C 180,E1 -5650.4,E2 -5650.4} C_VEL
LIN {X 0,Y 502.817,Z 291.853,A -85,B 0,C 180,E1 -5652.931,E2 -5652.931} C_VEL
LIN {X 0,Y 502.845,Z 291.849,A -85,B 0,C 180,E1 -5655.429,E2 -5655.429} C_VEL
LIN {X 0,Y 502.878,Z 291.847,A -85,B 0,C 180,E1 -5658.717,E2 -5658.717} C_VEL
LIN {X 0,Y 502.903,Z 291.84,A -85,B 0,C 180,E1 -5661.967,E2 -5661.967} C_VEL
LIN {X 0,Y 502.872,Z 291.849,A -85,B 0,C 180,E1 -5665.19,E2 -5665.19} C_VEL
LIN {X 0,Y 503.025,Z 291.828,A -85,B 0,C 180,E1 -5667.598,E2 -5667.598} C_VEL
LIN {X 0,Y 503.03,Z 291.825,A -85,B 0,C 180,E1 -5670,E2 -5670} C_VEL
LIN {X 0,Y 503.026,Z 291.827,A -85,B 0,C 180,E1 -5672.402,E2 -5672.402} C_VEL
LIN {X 0,Y 502.926,Z 291.84,A -85,B 0,C 180,E1 -5675.614,E2 -5675.614} C_VEL
LIN {X 0,Y 502.87,Z 291.846,A -85,B 0,C 180,E1 -5678.843,E2 -5678.843} C_VEL
LIN {X 0,Y 502.846,Z 291.849,A -85,B 0,C 180,E1 -5682.102,E2 -5682.102} C_VEL
LIN {X 0,Y 502.85,Z 291.848,A -85,B 0,C 180,E1 -5685.4,E2 -5685.4} C_VEL
LIN {X 0,Y 502.824,Z 291.854,A -85,B 0,C 180,E1 -5688.752,E2 -5688.752} C_VEL
LIN {X 0,Y 502.785,Z 291.857,A -85,B 0,C 180,E1 -5691.311,E2 -5691.311} C_VEL
LIN {X 0,Y 502.794,Z 291.856,A -85,B 0,C 180,E1 -5693.914,E2 -5693.914} C_VEL
LIN {X 0,Y 502.866,Z 291.849,A -85,B 0,C 180,E1 -5696.566,E2 -5696.566} C_VEL
LIN {X 0,Y 502.823,Z 291.853,A -85,B 0,C 180,E1 -5699.288,E2 -5699.288} C_VEL
LIN {X 0,Y 502.784,Z 291.86,A -85,B 0,C 180,E1 -5702.085,E2 -5702.085} C_VEL
LIN {X 0,Y 502.797,Z 291.855,A -85,B 0,C 180,E1 -5704.966,E2 -5704.966} C_VEL
LIN {X 0,Y 502.795,Z 291.856,A -85,B 0,C 180,E1 -5707.954,E2 -5707.954} C_VEL
LIN {X 0,Y 502.822,Z 291.853,A -85,B 0,C 180,E1 -5711.066,E2 -5711.066} C_VEL
LIN {X 0,Y 502.788,Z 291.856,A -85,B 0,C 180,E1 -5714.53,E2 -5714.53} C_VEL
LIN {X 0,Y 502.799,Z 291.857,A -85,B 0,C 180,E1 -5717.861,E2 -5717.861} C_VEL
LIN {X 0,Y 502.806,Z 291.854,A -85,B 0,C 180,E1 -5721.024,E2 -5721.024} C_VEL
LIN {X 0,Y 502.778,Z 291.86,A -85,B 0,C 180,E1 -5724.169,E2 -5724.169} C_VEL
LIN {X 0,Y 502.834,Z 291.852,A -85,B 0,C 180,E1 -5726.994,E2 -5726.994} C_VEL
LIN {X 0,Y 502.819,Z 291.852,A -85,B 0,C 180,E1 -5730.065,E2 -5730.065} C_VEL
LIN {X 0,Y 502.828,Z 291.852,A -85,B 0,C 180,E1 -5732.533,E2 -5732.533} C_VEL
LIN {X 0,Y 502.78,Z 291.858,A -85,B 0,C 180,E1 -5735.312,E2 -5735.312} C_VEL
LIN {X 0,Y 502.784,Z 291.857,A -85,B 0,C 180,E1 -5737.827,E2 -5737.827} C_VEL
LIN {X 0,Y 502.829,Z 291.852,A -85,B 0,C 180,E1 -5740.4,E2 -5740.4} C_VEL
LIN {X 0,Y 502.821,Z 291.854,A -85,B 0,C 180,E1 -5742.931,E2 -5742.931} C_VEL
LIN {X 0,Y 502.849,Z 291.851,A -85,B 0,C 180,E1 -5745.429,E2 -5745.429} C_VEL
LIN {X 0,Y 502.882,Z 291.844,A -85,B 0,C 180,E1 -5748.717,E2 -5748.717} C_VEL
LIN {X 0,Y 502.885,Z 291.845,A -85,B 0,C 180,E1 -5751.967,E2 -5751.967} C_VEL
LIN {X 0,Y 502.94,Z 291.838,A -85,B 0,C 180,E1 -5754.387,E2 -5754.387} C_VEL
LIN {X 0,Y 503.026,Z 291.826,A -85,B 0,C 180,E1 -5757.598,E2 -5757.598} C_VEL
LIN {X 0,Y 503.038,Z 291.826,A -85,B 0,C 180,E1 -5760.801,E2 -5760.801} C_VEL
LIN {X 0,Y 502.867,Z 291.847,A -85,B 0,C 180,E1 -5763.205,E2 -5763.205} C_VEL
LIN {X 0,Y 502.888,Z 291.846,A -85,B 0,C 180,E1 -5766.419,E2 -5766.419} C_VEL
LIN {X 0,Y 502.869,Z 291.849,A -85,B 0,C 180,E1 -5768.843,E2 -5768.843} C_VEL
LIN {X 0,Y 502.851,Z 291.849,A -85,B 0,C 180,E1 -5772.102,E2 -5772.102} C_VEL
LIN {X 0,Y 502.854,Z 291.849,A -85,B 0,C 180,E1 -5775.4,E2 -5775.4} C_VEL
LIN {X 0,Y 502.828,Z 291.851,A -85,B 0,C 180,E1 -5778.752,E2 -5778.752} C_VEL
LIN {X 0,Y 502.788,Z 291.855,A -85,B 0,C 180,E1 -5781.311,E2 -5781.311} C_VEL
LIN {X 0,Y 502.778,Z 291.858,A -85,B 0,C 180,E1 -5783.915,E2 -5783.915} C_VEL
LIN {X 0,Y 502.839,Z 291.85,A -85,B 0,C 180,E1 -5786.568,E2 -5786.568} C_VEL
LIN {X 0,Y 502.819,Z 291.854,A -85,B 0,C 180,E1 -5789.935,E2 -5789.935} C_VEL
LIN {X 0,Y 502.836,Z 291.849,A -85,B 0,C 180,E1 -5793.031,E2 -5793.031} C_VEL
LIN {X 0,Y 502.776,Z 291.858,A -85,B 0,C 180,E1 -5795.951,E2 -5795.951} C_VEL
LIN {X 0,Y 502.805,Z 291.855,A -85,B 0,C 180,E1 -5798.976,E2 -5798.976} C_VEL
LIN {X 0,Y 502.807,Z 291.854,A -85,B 0,C 180,E1 -5802.199,E2 -5802.199} C_VEL
LIN {X 0,Y 502.789,Z 291.856,A -85,B 0,C 180,E1 -5805.47,E2 -5805.47} C_VEL
LIN {X 0,Y 502.798,Z 291.854,A -85,B 0,C 180,E1 -5807.86,E2 -5807.86} C_VEL
LIN {X 0,Y 502.803,Z 291.883,A -85,B 0,C 180,E1 -5810.959,E2 -5810.959} C_VEL
LIN {X 0,Y 504.146,Z 299.136,A -85,B 0,C 180,E1 -5813.599,E2 -5813.599} C_VEL
LIN {X 0,Y 504.216,Z 304.225,A -85,B 0,C 180,E1 -5815.323,E2 -5815.323} C_VEL
LIN {X 0,Y 503.845,Z 313.409,A -85,B 0,C 180,E1 -5818.307,E2 -5818.307} C_VEL
LIN {X 0,Y 503.449,Z 324.134,A -85,B 0,C 180,E1 -5821.664,E2 -5821.664} C_VEL
LIN {X 0,Y 503.105,Z 334.443,A -85,B 0,C 180,E1 -5824.782,E2 -5824.782} C_VEL
LIN {X 0,Y 502.845,Z 344.784,A -85,B 0,C 180,E1 -5827.829,E2 -5827.829} C_VEL
LIN {X 0,Y 502.653,Z 355.199,A -85,B 0,C 180,E1 -5830.818,E2 -5830.818} C_VEL
LIN {X 0,Y 502.507,Z 365.556,A -85,B 0,C 180,E1 -5833.757,E2 -5833.757} C_VEL
LIN {X 0,Y 502.413,Z 372.4,A -85,B 0,C 180,E1 -5835.675,E2 -5835.675} C_VEL
LIN {X 0,Y 504.464,Z 387.401,A -85,B 0,C 180,E1 -5836.107,E2 -5836.107} C_VEL
LIN {X 0,Y 504.243,Z 400.417,A -85,B 0,C 180,E1 -5836.602,E2 -5836.602} C_VEL
LIN {X 0,Y 503.89,Z 412.038,A -85,B 0,C 180,E1 -5837.198,E2 -5837.198} C_VEL
LIN {X 0,Y 503.527,Z 422.971,A -85,B 0,C 180,E1 -5837.915,E2 -5837.915} C_VEL
LIN {X 0,Y 503.227,Z 433.997,A -85,B 0,C 180,E1 -5838.827,E2 -5838.827} C_VEL
LIN {X 0,Y 502.889,Z 442.975,A -85,B 0,C 180,E1 -5839.736,E2 -5839.736} C_VEL
LIN {X 0,Y 502.638,Z 452.739,A -85,B 0,C 180,E1 -5840.95,E2 -5840.95} C_VEL
LIN {X 0,Y 502.403,Z 460.526,A -85,B 0,C 180,E1 -5842.161,E2 -5842.161} C_VEL
LIN {X 0,Y 502.236,Z 467.285,A -85,B 0,C 180,E1 -5843.482,E2 -5843.482} C_VEL
LIN {X 0,Y 502.184,Z 472.475,A -85,B 0,C 180,E1 -5844.781,E2 -5844.781} C_VEL
LIN {X 0,Y 502.202,Z 476.128,A -85,B 0,C 180,E1 -5845.988,E2 -5845.988} C_VEL
LIN {X 0,Y 502.124,Z 478.005,A -85,B 0,C 180,E1 -5846.791,E2 -5846.791} C_VEL
LIN {X 0,Y 502.121,Z 479.416,A -85,B 0,C 180,E1 -5847.593,E2 -5847.593} C_VEL
LIN {X 0,Y 502.009,Z 481.021,A -85,B 0,C 180,E1 -5849.198,E2 -5849.198} C_VEL
LIN {X 0,Y 502.009,Z 481.232,A -85,B 0,C 180,E1 -5850,E2 -5850} C_VEL
LIN {X 0,Y 502.01,Z 481.007,A -85,B 0,C 180,E1 -5850.802,E2 -5850.802} C_VEL
LIN {X 0,Y 502.122,Z 479.373,A -85,B 0,C 180,E1 -5852.407,E2 -5852.407} C_VEL
LIN {X 0,Y 502.135,Z 477.946,A -85,B 0,C 180,E1 -5853.209,E2 -5853.209} C_VEL
LIN {X 0,Y 502.138,Z 474.952,A -85,B 0,C 180,E1 -5854.415,E2 -5854.415} C_VEL
LIN {X 0,Y 502.247,Z 470.91,A -85,B 0,C 180,E1 -5855.621,E2 -5855.621} C_VEL
LIN {X 0,Y 502.33,Z 464.794,A -85,B 0,C 180,E1 -5857.012,E2 -5857.012} C_VEL
LIN {X 0,Y 502.476,Z 457.902,A -85,B 0,C 180,E1 -5858.243,E2 -5858.243} C_VEL
LIN {X 0,Y 502.702,Z 449.485,A -85,B 0,C 180,E1 -5859.455,E2 -5859.455} C_VEL
LIN {X 0,Y 502.962,Z 440.858,A -85,B 0,C 180,E1 -5860.466,E2 -5860.466} C_VEL
LIN {X 0,Y 503.285,Z 430.219,A -85,B 0,C 180,E1 -5861.478,E2 -5861.478} C_VEL
LIN {X 0,Y 503.621,Z 418.788,A -85,B 0,C 180,E1 -5862.353,E2 -5862.353} C_VEL
LIN {X 0,Y 504.002,Z 408.205,A -85,B 0,C 180,E1 -5862.994,E2 -5862.994} C_VEL
LIN {X 0,Y 504.317,Z 396.367,A -85,B 0,C 180,E1 -5863.55,E2 -5863.55} C_VEL
LIN {X 0,Y 504.317,Z 386.838,A -85,B 0,C 180,E1 -5863.897,E2 -5863.897} C_VEL
LIN {X 0,Y 502.666,Z 374.266,A -85,B 0,C 180,E1 -5864.256,E2 -5864.256} C_VEL
LIN {X 0,Y 502.403,Z 371.878,A -85,B 0,C 180,E1 -5864.325,E2 -5864.325} C_VEL
LIN {X 0,Y 502.538,Z 360.342,A -85,B 0,C 180,E1 -5867.498,E2 -5867.498} C_VEL
LIN {X 0,Y 502.717,Z 348.259,A -85,B 0,C 180,E1 -5870.885,E2 -5870.885} C_VEL
LIN {X 0,Y 502.877,Z 337.766,A -85,B 0,C 180,E1 -5873.91,E2 -5873.91} C_VEL
LIN {X 0,Y 503.172,Z 327.306,A -85,B 0,C 180,E1 -5876.997,E2 -5876.997} C_VEL
LIN {X 0,Y 503.48,Z 316.982,A -85,B 0,C 180,E1 -5880.167,E2 -5880.167} C_VEL
LIN {X 0,Y 503.87,Z 306.679,A -85,B 0,C 180,E1 -5883.501,E2 -5883.501} C_VEL
LIN {X 0,Y 504.157,Z 299.869,A -85,B 0,C 180,E1 -5885.838,E2 -5885.838} C_VEL
LIN {X 0,Y 503.285,Z 294.36,A -85,B 0,C 180,E1 -5887.911,E2 -5887.911} C_VEL
LIN {X 0,Y 502.815,Z 291.852,A -85,B 0,C 180,E1 -5888.975,E2 -5888.975} C_VEL
LIN {X 0,Y 502.807,Z 291.857,A -85,B 0,C 180,E1 -5892.199,E2 -5892.199} C_VEL
LIN {X 0,Y 502.805,Z 291.858,A -85,B 0,C 180,E1 -5895.468,E2 -5895.468} C_VEL
LIN {X 0,Y 502.824,Z 291.856,A -85,B 0,C 180,E1 -5898.934,E2 -5898.934} C_VEL
LIN {X 0,Y 502.798,Z 291.858,A -85,B 0,C 180,E1 -5902.046,E2 -5902.046} C_VEL
LIN {X 0,Y 502.804,Z 291.856,A -85,B 0,C 180,E1 -5905.034,E2 -5905.034} C_VEL
LIN {X 0,Y 502.788,Z 291.858,A -85,B 0,C 180,E1 -5907.916,E2 -5907.916} C_VEL
LIN {X 0,Y 502.83,Z 291.852,A -85,B 0,C 180,E1 -5910.712,E2 -5910.712} C_VEL
LIN {X 0,Y 502.868,Z 291.848,A -85,B 0,C 180,E1 -5913.439,E2 -5913.439} C_VEL
LIN {X 0,Y 502.792,Z 291.858,A -85,B 0,C 180,E1 -5916.086,E2 -5916.086} C_VEL
LIN {X 0,Y 502.789,Z 291.857,A -85,B 0,C 180,E1 -5918.689,E2 -5918.689} C_VEL
LIN {X 0,Y 502.832,Z 291.853,A -85,B 0,C 180,E1 -5921.248,E2 -5921.248} C_VEL
LIN {X 0,Y 502.854,Z 291.848,A -85,B 0,C 180,E1 -5924.6,E2 -5924.6} C_VEL
LIN {X 0,Y 502.882,Z 291.847,A -85,B 0,C 180,E1 -5928.039,E2 -5928.039} C_VEL
LIN {X 0,Y 502.87,Z 291.848,A -85,B 0,C 180,E1 -5931.157,E2 -5931.157} C_VEL
LIN {X 0,Y 502.931,Z 291.84,A -85,B 0,C 180,E1 -5934.386,E2 -5934.386} C_VEL
LIN {X 0,Y 503.03,Z 291.827,A -85,B 0,C 180,E1 -5937.598,E2 -5937.598} C_VEL
LIN {X 0,Y 503.034,Z 291.828,A -85,B 0,C 180,E1 -5940,E2 -5940} C_VEL
LIN {X 0,Y 503.031,Z 291.828,A -85,B 0,C 180,E1 -5942.402,E2 -5942.402} C_VEL
LIN {X 0,Y 502.933,Z 291.84,A -85,B 0,C 180,E1 -5945.613,E2 -5945.613} C_VEL
LIN {X 0,Y 502.874,Z 291.848,A -85,B 0,C 180,E1 -5948.034,E2 -5948.034} C_VEL
LIN {X 0,Y 502.623,Z 291.881,A -85,B 0,C 180,E1 -5951.289,E2 -5951.289} C_VEL
LIN {X 0,Y 502.514,Z 292.064,A -85,B 0,C 180,E1 -5952.11,E2 -5952.11} C_VEL
LIN {X 0,Y 502.449,Z 295.242,A -85,B 0,C 180,E1 -5955.412,E2 -5955.412} C_VEL
LIN {X 0,Y 502.315,Z 298.589,A -85,B 0,C 180,E1 -5958.772,E2 -5958.772} C_VEL
LIN {X 0,Y 502.281,Z 301.09,A -85,B 0,C 180,E1 -5961.333,E2 -5961.333} C_VEL
LIN {X 0,Y 502.273,Z 303.608,A -85,B 0,C 180,E1 -5963.83,E2 -5963.83} C_VEL
LIN {X 0,Y 504.727,Z 314.39,A -85,B 0,C 180,E1 -5964.2,E2 -5964.2} C_VEL
LIN {X 0,Y 504.518,Z 327.171,A -85,B 0,C 180,E1 -5964.702,E2 -5964.702} C_VEL
LIN {X 0,Y 504.219,Z 339.275,A -85,B 0,C 180,E1 -5965.347,E2 -5965.347} C_VEL
LIN {X 0,Y 503.814,Z 351.15,A -85,B 0,C 180,E1 -5966.178,E2 -5966.178} C_VEL
LIN {X 0,Y 503.455,Z 362.002,A -85,B 0,C 180,E1 -5967.136,E2 -5967.136} C_VEL
LIN {X 0,Y 503.157,Z 370.992,A -85,B 0,C 180,E1 -5968.121,E2 -5968.121} C_VEL
LIN {X 0,Y 502.869,Z 379.596,A -85,B 0,C 180,E1 -5969.285,E2 -5969.285} C_VEL
LIN {X 0,Y 502.625,Z 386.614,A -85,B 0,C 180,E1 -5970.455,E2 -5970.455} C_VEL
LIN {X 0,Y 502.432,Z 392.777,A -85,B 0,C 180,E1 -5971.74,E2 -5971.74} C_VEL
LIN {X 0,Y 502.295,Z 397.689,A -85,B 0,C 180,E1 -5973.071,E2 -5973.071} C_VEL
LIN {X 0,Y 502.178,Z 401.162,A -85,B 0,C 180,E1 -5974.339,E2 -5974.339} C_VEL
LIN {X 0,Y 502.081,Z 403.714,A -85,B 0,C 180,E1 -5975.72,E2 -5975.72} C_VEL
LIN {X 0,Y 502.041,Z 405.051,A -85,B 0,C 180,E1 -5977.066,E2 -5977.066} C_VEL
LIN {X 0,Y 502.023,Z 405.292,A -85,B 0,C 180,E1 -5978.374,E2 -5978.374} C_VEL
LIN {X 0,Y 502.067,Z 404.516,A -85,B 0,C 180,E1 -5979.655,E2 -5979.655} C_VEL
LIN {X 0,Y 502.149,Z 402.372,A -85,B 0,C 180,E1 -5981.133,E2 -5981.133} C_VEL
LIN {X 0,Y 502.261,Z 399.942,A -85,B 0,C 180,E1 -5982.195,E2 -5982.195} C_VEL
LIN {X 0,Y 502.357,Z 396.523,A -85,B 0,C 180,E1 -5983.324,E2 -5983.324} C_VEL
LIN {X 0,Y 502.465,Z 391.088,A -85,B 0,C 180,E1 -5984.69,E2 -5984.69} C_VEL
LIN {X 0,Y 502.605,Z 385.312,A -85,B 0,C 180,E1 -5985.833,E2 -5985.833} C_VEL
LIN {X 0,Y 502.892,Z 377.761,A -85,B 0,C 180,E1 -5987.041,E2 -5987.041} C_VEL
LIN {X 0,Y 503.125,Z 369.048,A -85,B 0,C 180,E1 -5988.163,E2 -5988.163} C_VEL
LIN {X 0,Y 503.541,Z 358.363,A -85,B 0,C 180,E1 -5989.269,E2 -5989.269} C_VEL
LIN {X 0,Y 503.89,Z 347.336,A -85,B 0,C 180,E1 -5990.175,E2 -5990.175} C_VEL
LIN {X 0,Y 503.441,Z 342.399,A -85,B 0,C 180,E1 -5990.537,E2 -5990.537} C_VEL
LIN {X 0,Y 501.012,Z 334.199,A -85,B 0,C 180,E1 -5991.113,E2 -5991.113} C_VEL
LIN {X 0,Y 498.433,Z 325.731,A -85,B 0,C 180,E1 -5991.62,E2 -5991.62} C_VEL
LIN {X 0,Y 497.789,Z 320.293,A -85,B 0,C 180,E1 -5991.87,E2 -5991.87} C_VEL
LIN {X 0,Y 497.616,Z 314.324,A -85,B 0,C 180,E1 -5992.094,E2 -5992.094} C_VEL
LIN {X 0,Y 495.086,Z 303.277,A -85,B 0,C 180,E1 -5992.485,E2 -5992.485} C_VEL
LIN {X 0,Y 495.12,Z 300.181,A -85,B 0,C 180,E1 -5995.415,E2 -5995.415} C_VEL
LIN {X 0,Y 495.154,Z 297.072,A -85,B 0,C 180,E1 -5998.388,E2 -5998.388} C_VEL
LIN {X 0,Y 495.212,Z 294.176,A -85,B 0,C 180,E1 -6001.149,E2 -6001.149} C_VEL
LIN {X 0,Y 495.233,Z 293.21,A -85,B 0,C 180,E1 -6002.075,E2 -6002.075} C_VEL
LIN {X 0,Y 495.329,Z 292.788,A -85,B 0,C 180,E1 -6003.365,E2 -6003.365} C_VEL
LIN {X 0,Y 495.566,Z 292.758,A -85,B 0,C 180,E1 -6005.715,E2 -6005.715} C_VEL
LIN {X 0,Y 495.735,Z 292.735,A -85,B 0,C 180,E1 -6007.494,E2 -6007.494} C_VEL
LIN {X 0,Y 495.77,Z 292.729,A -85,B 0,C 180,E1 -6010.109,E2 -6010.109} C_VEL
LIN {X 0,Y 495.762,Z 292.732,A -85,B 0,C 180,E1 -6012.68,E2 -6012.68} C_VEL
LIN {X 0,Y 495.791,Z 292.728,A -85,B 0,C 180,E1 -6015.217,E2 -6015.217} C_VEL
LIN {X 0,Y 495.853,Z 292.721,A -85,B 0,C 180,E1 -6018.555,E2 -6018.555} C_VEL
LIN {X 0,Y 495.874,Z 292.716,A -85,B 0,C 180,E1 -6021.852,E2 -6021.852} C_VEL
LIN {X 0,Y 495.84,Z 292.724,A -85,B 0,C 180,E1 -6025.121,E2 -6025.121} C_VEL
LIN {X 0,Y 495.994,Z 292.703,A -85,B 0,C 180,E1 -6027.564,E2 -6027.564} C_VEL
LIN {X 0,Y 496.001,Z 292.7,A -85,B 0,C 180,E1 -6030,E2 -6030} C_VEL
LIN {X 0,Y 495.995,Z 292.703,A -85,B 0,C 180,E1 -6032.436,E2 -6032.436} C_VEL
LIN {X 0,Y 495.881,Z 292.717,A -85,B 0,C 180,E1 -6035.694,E2 -6035.694} C_VEL
LIN {X 0,Y 495.839,Z 292.722,A -85,B 0,C 180,E1 -6038.97,E2 -6038.97} C_VEL
LIN {X 0,Y 495.83,Z 292.723,A -85,B 0,C 180,E1 -6042.035,E2 -6042.035} C_VEL
LIN {X 0,Y 495.825,Z 292.723,A -85,B 0,C 180,E1 -6045.452,E2 -6045.452} C_VEL
LIN {X 0,Y 495.78,Z 292.73,A -85,B 0,C 180,E1 -6049.029,E2 -6049.029} C_VEL
LIN {X 0,Y 495.745,Z 292.735,A -85,B 0,C 180,E1 -6051.629,E2 -6051.629} C_VEL
LIN {X 0,Y 495.782,Z 292.729,A -85,B 0,C 180,E1 -6054.874,E2 -6054.874} C_VEL
LIN {X 0,Y 495.814,Z 292.725,A -85,B 0,C 180,E1 -6056.974,E2 -6056.974} C_VEL
LIN {X 0,Y 495.764,Z 292.732,A -85,B 0,C 180,E1 -6060.147,E2 -6060.147} C_VEL
LIN {X 0,Y 495.791,Z 292.729,A -85,B 0,C 180,E1 -6063.244,E2 -6063.244} C_VEL
LIN {X 0,Y 495.721,Z 292.739,A -85,B 0,C 180,E1 -6066.089,E2 -6066.089} C_VEL
LIN {X 0,Y 495.766,Z 292.731,A -85,B 0,C 180,E1 -6068.769,E2 -6068.769} C_VEL
LIN {X 0,Y 495.758,Z 292.732,A -85,B 0,C 180,E1 -6071.781,E2 -6071.781} C_VEL
LIN {X 0,Y 495.739,Z 292.735,A -85,B 0,C 180,E1 -6075.141,E2 -6075.141} C_VEL
LIN {X 0,Y 495.76,Z 292.731,A -85,B 0,C 180,E1 -6078.219,E2 -6078.219} C_VEL
LIN {X 0,Y 495.754,Z 292.733,A -85,B 0,C 180,E1 -6081.409,E2 -6081.409} C_VEL
LIN {X 0,Y 495.75,Z 292.734,A -85,B 0,C 180,E1 -6084.463,E2 -6084.463} C_VEL
LIN {X 0,Y 495.769,Z 292.731,A -85,B 0,C 180,E1 -6087.406,E2 -6087.406} C_VEL
LIN {X 0,Y 495.769,Z 292.729,A -85,B 0,C 180,E1 -6090.254,E2 -6090.254} C_VEL
LIN {X 0,Y 495.809,Z 292.726,A -85,B 0,C 180,E1 -6093.255,E2 -6093.255} C_VEL
LIN {X 0,Y 495.744,Z 292.734,A -85,B 0,C 180,E1 -6096.613,E2 -6096.613} C_VEL
LIN {X 0,Y 495.783,Z 292.729,A -85,B 0,C 180,E1 -6099.324,E2 -6099.324} C_VEL
LIN {X 0,Y 495.786,Z 292.728,A -85,B 0,C 180,E1 -6101.829,E2 -6101.829} C_VEL
LIN {X 0,Y 495.829,Z 292.723,A -85,B 0,C 180,E1 -6104.549,E2 -6104.549} C_VEL
LIN {X 0,Y 495.834,Z 292.724,A -85,B 0,C 180,E1 -6107.965,E2 -6107.965} C_VEL
LIN {X 0,Y 495.839,Z 292.723,A -85,B 0,C 180,E1 -6111.03,E2 -6111.03} C_VEL
LIN {X 0,Y 495.885,Z 292.716,A -85,B 0,C 180,E1 -6113.49,E2 -6113.49} C_VEL
LIN {X 0,Y 495.824,Z 292.724,A -85,B 0,C 180,E1 -6116.75,E2 -6116.75} C_VEL
LIN {X 0,Y 495.875,Z 292.718,A -85,B 0,C 180,E1 -6118.376,E2 -6118.376} C_VEL
LIN {X 0,Y 495.988,Z 292.704,A -85,B 0,C 180,E1 -6120.812,E2 -6120.812} C_VEL
LIN {X 0,Y 495.99,Z 292.705,A -85,B 0,C 180,E1 -6122.436,E2 -6122.436} C_VEL
LIN {X 0,Y 495.886,Z 292.714,A -85,B 0,C 180,E1 -6125.694,E2 -6125.694} C_VEL
LIN {X 0,Y 495.839,Z 292.724,A -85,B 0,C 180,E1 -6128.97,E2 -6128.97} C_VEL
LIN {X 0,Y 495.834,Z 292.723,A -85,B 0,C 180,E1 -6132.035,E2 -6132.035} C_VEL
LIN {X 0,Y 495.829,Z 292.724,A -85,B 0,C 180,E1 -6135.451,E2 -6135.451} C_VEL
LIN {X 0,Y 495.784,Z 292.729,A -85,B 0,C 180,E1 -6139.029,E2 -6139.029} C_VEL
LIN {X 0,Y 495.747,Z 292.732,A -85,B 0,C 180,E1 -6141.629,E2 -6141.629} C_VEL
LIN {X 0,Y 495.726,Z 292.736,A -85,B 0,C 180,E1 -6144.277,E2 -6144.277} C_VEL
LIN {X 0,Y 495.763,Z 292.732,A -85,B 0,C 180,E1 -6146.977,E2 -6146.977} C_VEL
LIN {X 0,Y 495.768,Z 292.733,A -85,B 0,C 180,E1 -6150.147,E2 -6150.147} C_VEL
LIN {X 0,Y 495.797,Z 292.725,A -85,B 0,C 180,E1 -6153.244,E2 -6153.244} C_VEL
LIN {X 0,Y 495.722,Z 292.737,A -85,B 0,C 180,E1 -6156.088,E2 -6156.088} C_VEL
LIN {X 0,Y 495.767,Z 292.731,A -85,B 0,C 180,E1 -6158.768,E2 -6158.768} C_VEL
LIN {X 0,Y 495.754,Z 292.735,A -85,B 0,C 180,E1 -6161.782,E2 -6161.782} C_VEL
LIN {X 0,Y 495.741,Z 292.733,A -85,B 0,C 180,E1 -6165.141,E2 -6165.141} C_VEL
LIN {X 0,Y 495.754,Z 292.734,A -85,B 0,C 180,E1 -6168.218,E2 -6168.218} C_VEL
LIN {X 0,Y 495.77,Z 292.747,A -85,B 0,C 180,E1 -6170.704,E2 -6170.704} C_VEL
LIN {X 0,Y 497.223,Z 300.793,A -85,B 0,C 180,E1 -6173.675,E2 -6173.675} C_VEL
LIN {X 0,Y 497.186,Z 306.328,A -85,B 0,C 180,E1 -6175.568,E2 -6175.568} C_VEL
LIN {X 0,Y 496.807,Z 315.054,A -85,B 0,C 180,E1 -6178.438,E2 -6178.438} C_VEL
LIN {X 0,Y 496.413,Z 325.509,A -85,B 0,C 180,E1 -6181.759,E2 -6181.759} C_VEL
LIN {X 0,Y 496.06,Z 336.254,A -85,B 0,C 180,E1 -6185.058,E2 -6185.058} C_VEL
LIN {X 0,Y 495.734,Z 347.379,A -85,B 0,C 180,E1 -6188.37,E2 -6188.37} C_VEL
LIN {X 0,Y 495.584,Z 357.717,A -85,B 0,C 180,E1 -6191.393,E2 -6191.393} C_VEL
LIN {X 0,Y 495.356,Z 369.4,A -85,B 0,C 180,E1 -6194.747,E2 -6194.747} C_VEL
LIN {X 0,Y 495.314,Z 371.913,A -85,B 0,C 180,E1 -6195.465,E2 -6195.465} C_VEL
LIN {X 0,Y 497.383,Z 387.203,A -85,B 0,C 180,E1 -6195.918,E2 -6195.918} C_VEL
LIN {X 0,Y 497.425,Z 395.029,A -85,B 0,C 180,E1 -6196.206,E2 -6196.206} C_VEL
LIN {X 0,Y 497.073,Z 408.099,A -85,B 0,C 180,E1 -6196.821,E2 -6196.821} C_VEL
LIN {X 0,Y 496.633,Z 419.582,A -85,B 0,C 180,E1 -6197.539,E2 -6197.539} C_VEL
LIN {X 0,Y 496.286,Z 431.199,A -85,B 0,C 180,E1 -6198.461,E2 -6198.461} C_VEL
LIN {X 0,Y 495.952,Z 440.605,A -85,B 0,C 180,E1 -6199.384,E2 -6199.384} C_VEL
LIN {X 0,Y 495.628,Z 449.19,A -85,B 0,C 180,E1 -6200.409,E2 -6200.409} C_VEL
LIN {X 0,Y 495.428,Z 457.563,A -85,B 0,C 180,E1 -6201.639,E2 -6201.639} C_VEL
LIN {X 0,Y 495.26,Z 464.314,A -85,B 0,C 180,E1 -6202.867,E2 -6202.867} C_VEL
LIN {X 0,Y 495.157,Z 470.501,A -85,B 0,C 180,E1 -6204.298,E2 -6204.298} C_VEL
LIN {X 0,Y 495.027,Z 474.51,A -85,B 0,C 180,E1 -6205.521,E2 -6205.521} C_VEL
LIN {X 0,Y 495.048,Z 477.475,A -85,B 0,C 180,E1 -6206.745,E2 -6206.745} C_VEL
LIN {X 0,Y 495.054,Z 478.888,A -85,B 0,C 180,E1 -6207.559,E2 -6207.559} C_VEL
LIN {X 0,Y 494.928,Z 480.488,A -85,B 0,C 180,E1 -6209.186,E2 -6209.186} C_VEL
LIN {X 0,Y 494.929,Z 480.698,A -85,B 0,C 180,E1 -6210,E2 -6210} C_VEL
LIN {X 0,Y 494.93,Z 480.47,A -85,B 0,C 180,E1 -6210.814,E2 -6210.814} C_VEL
LIN {X 0,Y 495.055,Z 478.83,A -85,B 0,C 180,E1 -6212.441,E2 -6212.441} C_VEL
LIN {X 0,Y 495.059,Z 477.398,A -85,B 0,C 180,E1 -6213.255,E2 -6213.255} C_VEL
LIN {X 0,Y 495.04,Z 474.394,A -85,B 0,C 180,E1 -6214.478,E2 -6214.478} C_VEL
LIN {X 0,Y 495.158,Z 470.344,A -85,B 0,C 180,E1 -6215.702,E2 -6215.702} C_VEL
LIN {X 0,Y 495.256,Z 464.113,A -85,B 0,C 180,E1 -6217.133,E2 -6217.133} C_VEL
LIN {X 0,Y 495.399,Z 457.309,A -85,B 0,C 180,E1 -6218.361,E2 -6218.361} C_VEL
LIN {X 0,Y 495.626,Z 448.879,A -85,B 0,C 180,E1 -6219.591,E2 -6219.591} C_VEL
LIN {X 0,Y 495.937,Z 440.24,A -85,B 0,C 180,E1 -6220.616,E2 -6220.616} C_VEL
LIN {X 0,Y 496.307,Z 429.589,A -85,B 0,C 180,E1 -6221.642,E2 -6221.642} C_VEL
LIN {X 0,Y 496.613,Z 418.054,A -85,B 0,C 180,E1 -6222.536,E2 -6222.536} C_VEL
LIN {X 0,Y 497.06,Z 405.568,A -85,B 0,C 180,E1 -6223.283,E2 -6223.283} C_VEL
LIN {X 0,Y 497.445,Z 393.105,A -85,B 0,C 180,E1 -6223.845,E2 -6223.845} C_VEL
LIN {X 0,Y 497.345,Z 387.302,A -85,B 0,C 180,E1 -6224.057,E2 -6224.057} C_VEL
LIN {X 0,Y 495.694,Z 374.475,A -85,B 0,C 180,E1 -6224.445,E2 -6224.445} C_VEL
LIN {X 0,Y 495.303,Z 371.268,A -85,B 0,C 180,E1 -6224.535,E2 -6224.535} C_VEL
LIN {X 0,Y 495.447,Z 361.307,A -85,B 0,C 180,E1 -6227.331,E2 -6227.331} C_VEL
LIN {X 0,Y 495.646,Z 349.254,A -85,B 0,C 180,E1 -6230.762,E2 -6230.762} C_VEL
LIN {X 0,Y 495.814,Z 338.816,A -85,B 0,C 180,E1 -6233.827,E2 -6233.827} C_VEL
LIN {X 0,Y 496.12,Z 328.316,A -85,B 0,C 180,E1 -6236.957,E2 -6236.957} C_VEL
LIN {X 0,Y 496.471,Z 317.738,A -85,B 0,C 180,E1 -6240.286,E2 -6240.286} C_VEL
LIN {X 0,Y 496.884,Z 308.069,A -85,B 0,C 180,E1 -6243.479,E2 -6243.479} C_VEL
LIN {X 0,Y 497.191,Z 301.25,A -85,B 0,C 180,E1 -6245.854,E2 -6245.854} C_VEL
LIN {X 0,Y 496.297,Z 295.596,A -85,B 0,C 180,E1 -6248.024,E2 -6248.024} C_VEL
LIN {X 0,Y 495.752,Z 292.731,A -85,B 0,C 180,E1 -6249.234,E2 -6249.234} C_VEL
LIN {X 0,Y 495.76,Z 292.734,A -85,B 0,C 180,E1 -6251.781,E2 -6251.781} C_VEL
LIN {X 0,Y 495.754,Z 292.738,A -85,B 0,C 180,E1 -6255.139,E2 -6255.139} C_VEL
LIN {X 0,Y 495.76,Z 292.736,A -85,B 0,C 180,E1 -6258.219,E2 -6258.219} C_VEL
LIN {X 0,Y 495.756,Z 292.734,A -85,B 0,C 180,E1 -6261.409,E2 -6261.409} C_VEL
LIN {X 0,Y 495.753,Z 292.734,A -85,B 0,C 180,E1 -6264.462,E2 -6264.462} C_VEL
LIN {X 0,Y 495.772,Z 292.732,A -85,B 0,C 180,E1 -6267.406,E2 -6267.406} C_VEL
LIN {X 0,Y 495.772,Z 292.732,A -85,B 0,C 180,E1 -6270.254,E2 -6270.254} C_VEL
LIN {X 0,Y 495.829,Z 292.725,A -85,B 0,C 180,E1 -6273.251,E2 -6273.251} C_VEL
LIN {X 0,Y 495.754,Z 292.732,A -85,B 0,C 180,E1 -6275.725,E2 -6275.725} C_VEL
LIN {X 0,Y 495.748,Z 292.735,A -85,B 0,C 180,E1 -6278.371,E2 -6278.371} C_VEL
LIN {X 0,Y 495.788,Z 292.73,A -85,B 0,C 180,E1 -6280.972,E2 -6280.972} C_VEL
LIN {X 0,Y 495.813,Z 292.725,A -85,B 0,C 180,E1 -6284.376,E2 -6284.376} C_VEL
LIN {X 0,Y 495.789,Z 292.728,A -85,B 0,C 180,E1 -6286.891,E2 -6286.891} C_VEL
LIN {X 0,Y 495.78,Z 292.731,A -85,B 0,C 180,E1 -6289.381,E2 -6289.381} C_VEL
LIN {X 0,Y 495.836,Z 292.723,A -85,B 0,C 180,E1 -6291.851,E2 -6291.851} C_VEL
LIN {X 0,Y 495.842,Z 292.723,A -85,B 0,C 180,E1 -6295.121,E2 -6295.121} C_VEL
LIN {X 0,Y 495.999,Z 292.703,A -85,B 0,C 180,E1 -6297.564,E2 -6297.564} C_VEL
LIN {X 0,Y 495.989,Z 292.704,A -85,B 0,C 180,E1 -6300.812,E2 -6300.812} C_VEL
LIN {X 0,Y 495.999,Z 292.704,A -85,B 0,C 180,E1 -6302.436,E2 -6302.436} C_VEL
LIN {X 0,Y 495.888,Z 292.717,A -85,B 0,C 180,E1 -6305.693,E2 -6305.693} C_VEL
LIN {X 0,Y 495.828,Z 292.727,A -85,B 0,C 180,E1 -6308.149,E2 -6308.149} C_VEL
LIN {X 0,Y 495.574,Z 292.758,A -85,B 0,C 180,E1 -6311.452,E2 -6311.452} C_VEL
LIN {X 0,Y 495.44,Z 293.052,A -85,B 0,C 180,E1 -6312.285,E2 -6312.285} C_VEL
LIN {X 0,Y 495.418,Z 295.968,A -85,B 0,C 180,E1 -6315.279,E2 -6315.279} C_VEL
LIN {X 0,Y 495.277,Z 298.808,A -85,B 0,C 180,E1 -6318.191,E2 -6318.191} C_VEL
LIN {X 0,Y 495.251,Z 301.333,A -85,B 0,C 180,E1 -6320.779,E2 -6320.779} C_VEL
LIN {X 0,Y 495.19,Z 304.128,A -85,B 0,C 180,E1 -6323.609,E2 -6323.609} C_VEL
LIN {X 0,Y 497.856,Z 315.549,A -85,B 0,C 180,E1 -6324.027,E2 -6324.027} C_VEL
LIN {X 0,Y 497.625,Z 328.796,A -85,B 0,C 180,E1 -6324.566,E2 -6324.566} C_VEL
LIN {X 0,Y 497.28,Z 340.941,A -85,B 0,C 180,E1 -6325.242,E2 -6325.242} C_VEL
LIN {X 0,Y 496.827,Z 353.068,A -85,B 0,C 180,E1 -6326.122,E2 -6326.122} C_VEL
LIN {X 0,Y 496.487,Z 363.194,A -85,B 0,C 180,E1 -6327.048,E2 -6327.048} C_VEL
LIN {X 0,Y 496.159,Z 372.262,A -85,B 0,C 180,E1 -6328.075,E2 -6328.075} C_VEL
LIN {X 0,Y 495.842,Z 380.876,A -85,B 0,C 180,E1 -6329.275,E2 -6329.275} C_VEL
LIN {X 0,Y 495.605,Z 387.284,A -85,B 0,C 180,E1 -6330.372,E2 -6330.372} C_VEL
LIN {X 0,Y 495.415,Z 393.359,A -85,B 0,C 180,E1 -6331.66,E2 -6331.66} C_VEL
LIN {X 0,Y 495.218,Z 398.656,A -85,B 0,C 180,E1 -6333.142,E2 -6333.142} C_VEL
LIN {X 0,Y 495.077,Z 402.376,A -85,B 0,C 180,E1 -6334.599,E2 -6334.599} C_VEL
LIN {X 0,Y 494.99,Z 404.635,A -85,B 0,C 180,E1 -6335.972,E2 -6335.972} C_VEL
LIN {X 0,Y 494.948,Z 405.743,A -85,B 0,C 180,E1 -6337.328,E2 -6337.328} C_VEL
LIN {X 0,Y 494.972,Z 405.761,A -85,B 0,C 180,E1 -6338.664,E2 -6338.664} C_VEL
LIN {X 0,Y 494.999,Z 404.782,A -85,B 0,C 180,E1 -6339.942,E2 -6339.942} C_VEL
LIN {X 0,Y 495.08,Z 402.847,A -85,B 0,C 180,E1 -6341.203,E2 -6341.203} C_VEL
LIN {X 0,Y 495.211,Z 399.974,A -85,B 0,C 180,E1 -6342.44,E2 -6342.44} C_VEL
LIN {X 0,Y 495.3,Z 396.19,A -85,B 0,C 180,E1 -6343.642,E2 -6343.642} C_VEL
LIN {X 0,Y 495.435,Z 391.42,A -85,B 0,C 180,E1 -6344.823,E2 -6344.823} C_VEL
LIN {X 0,Y 495.589,Z 385.599,A -85,B 0,C 180,E1 -6345.982,E2 -6345.982} C_VEL
LIN {X 0,Y 495.875,Z 378.496,A -85,B 0,C 180,E1 -6347.132,E2 -6347.132} C_VEL
LIN {X 0,Y 496.149,Z 369.931,A -85,B 0,C 180,E1 -6348.259,E2 -6348.259} C_VEL
LIN {X 0,Y 496.57,Z 359.333,A -85,B 0,C 180,E1 -6349.379,E2 -6349.379} C_VEL
LIN {X 0,Y 496.949,Z 348.188,A -85,B 0,C 180,E1 -6350.317,E2 -6350.317} C_VEL
LIN {X 0,Y 497.329,Z 336.586,A -85,B 0,C 180,E1 -6351.084,E2 -6351.084} C_VEL
LIN {X 0,Y 497.711,Z 324.094,A -85,B 0,C 180,E1 -6351.717,E2 -6351.717} C_VEL
LIN {X 0,Y 497.789,Z 320.293,A -85,B 0,C 180,E1 -6351.87,E2 -6351.87} C_VEL
LIN {X 0,Y 497.074,Z 318.434,A -85,B 0,C 180,E1 -6351.967,E2 -6351.967} C_VEL
LIN {X 0,Y 494.268,Z 316.251,A -85,B 0,C 180,E1 -6352.137,E2 -6352.137} C_VEL
LIN {X 0,Y 490.936,Z 313.841,A -85,B 0,C 180,E1 -6352.32,E2 -6352.32} C_VEL
LIN {X 0,Y 490.086,Z 312.245,A -85,B 0,C 180,E1 -6352.395,E2 -6352.395} C_VEL
LIN {X 0,Y 488.043,Z 303.745,A -85,B 0,C 180,E1 -6352.697,E2 -6352.697} C_VEL
LIN {X 0,Y 488.06,Z 300.424,A -85,B 0,C 180,E1 -6355.834,E2 -6355.834} C_VEL
LIN {X 0,Y 488.084,Z 297.334,A -85,B 0,C 180,E1 -6358.777,E2 -6358.777} C_VEL
LIN {X 0,Y 488.18,Z 294.338,A -85,B 0,C 180,E1 -6361.635,E2 -6361.635} C_VEL
LIN {X 0,Y 488.182,Z 293.68,A -85,B 0,C 180,E1 -6362.569,E2 -6362.569} C_VEL
LIN {X 0,Y 488.521,Z 293.637,A -85,B 0,C 180,E1 -6365.342,E2 -6365.342} C_VEL
LIN {X 0,Y 488.719,Z 293.611,A -85,B 0,C 180,E1 -6367.153,E2 -6367.153} C_VEL
LIN {X 0,Y 488.725,Z 293.607,A -85,B 0,C 180,E1 -6369.81,E2 -6369.81} C_VEL
LIN {X 0,Y 488.713,Z 293.611,A -85,B 0,C 180,E1 -6372.422,E2 -6372.422} C_VEL
LIN {X 0,Y 488.763,Z 293.605,A -85,B 0,C 180,E1 -6375,E2 -6375} C_VEL
LIN {X 0,Y 488.807,Z 293.597,A -85,B 0,C 180,E1 -6378.387,E2 -6378.387} C_VEL
LIN {X 0,Y 488.818,Z 293.595,A -85,B 0,C 180,E1 -6381.734,E2 -6381.734} C_VEL
LIN {X 0,Y 488.809,Z 293.599,A -85,B 0,C 180,E1 -6385.051,E2 -6385.051} C_VEL
LIN {X 0,Y 488.962,Z 293.579,A -85,B 0,C 180,E1 -6387.529,E2 -6387.529} C_VEL
LIN {X 0,Y 488.972,Z 293.576,A -85,B 0,C 180,E1 -6390,E2 -6390} C_VEL
LIN {X 0,Y 488.963,Z 293.579,A -85,B 0,C 180,E1 -6392.471,E2 -6392.471} C_VEL
LIN {X 0,Y 488.839,Z 293.595,A -85,B 0,C 180,E1 -6395.776,E2 -6395.776} C_VEL
LIN {X 0,Y 488.817,Z 293.598,A -85,B 0,C 180,E1 -6398.266,E2 -6398.266} C_VEL
LIN {X 0,Y 488.807,Z 293.597,A -85,B 0,C 180,E1 -6401.613,E2 -6401.613} C_VEL
LIN {X 0,Y 488.761,Z 293.605,A -85,B 0,C 180,E1 -6405.001,E2 -6405.001} C_VEL
LIN {X 0,Y 488.747,Z 293.606,A -85,B 0,C 180,E1 -6408.443,E2 -6408.443} C_VEL
LIN {X 0,Y 488.709,Z 293.61,A -85,B 0,C 180,E1 -6411.071,E2 -6411.071} C_VEL
LIN {X 0,Y 488.695,Z 293.611,A -85,B 0,C 180,E1 -6413.746,E2 -6413.746} C_VEL
LIN {X 0,Y 488.793,Z 293.6,A -85,B 0,C 180,E1 -6416.944,E2 -6416.944} C_VEL
LIN {X 0,Y 488.709,Z 293.611,A -85,B 0,C 180,E1 -6420.363,E2 -6420.363} C_VEL
LIN {X 0,Y 488.731,Z 293.609,A -85,B 0,C 180,E1 -6423.483,E2 -6423.483} C_VEL
LIN {X 0,Y 488.684,Z 293.613,A -85,B 0,C 180,E1 -6426.355,E2 -6426.355} C_VEL
LIN {X 0,Y 488.703,Z 293.61,A -85,B 0,C 180,E1 -6429.254,E2 -6429.254} C_VEL
LIN {X 0,Y 488.709,Z 293.611,A -85,B 0,C 180,E1 -6431.6,E2 -6431.6} C_VEL
LIN {X 0,Y 488.704,Z 293.611,A -85,B 0,C 180,E1 -6434.803,E2 -6434.803} C_VEL
LIN {X 0,Y 488.694,Z 293.612,A -85,B 0,C 180,E1 -6437.475,E2 -6437.475} C_VEL
LIN {X 0,Y 488.736,Z 293.607,A -85,B 0,C 180,E1 -6439.677,E2 -6439.677} C_VEL
LIN {X 0,Y 488.683,Z 293.613,A -85,B 0,C 180,E1 -6442.841,E2 -6442.841} C_VEL
LIN {X 0,Y 488.727,Z 293.609,A -85,B 0,C 180,E1 -6445.887,E2 -6445.887} C_VEL
LIN {X 0,Y 488.695,Z 293.611,A -85,B 0,C 180,E1 -6448.821,E2 -6448.821} C_VEL
LIN {X 0,Y 488.745,Z 293.606,A -85,B 0,C 180,E1 -6451.671,E2 -6451.671} C_VEL
LIN {X 0,Y 488.714,Z 293.609,A -85,B 0,C 180,E1 -6454.442,E2 -6454.442} C_VEL
LIN {X 0,Y 488.726,Z 293.609,A -85,B 0,C 180,E1 -6457.153,E2 -6457.153} C_VEL
LIN {X 0,Y 488.73,Z 293.609,A -85,B 0,C 180,E1 -6459.811,E2 -6459.811} C_VEL
LIN {X 0,Y 488.718,Z 293.608,A -85,B 0,C 180,E1 -6462.423,E2 -6462.423} C_VEL
LIN {X 0,Y 488.766,Z 293.603,A -85,B 0,C 180,E1 -6465,E2 -6465} C_VEL
LIN {X 0,Y 488.811,Z 293.598,A -85,B 0,C 180,E1 -6468.388,E2 -6468.388} C_VEL
LIN {X 0,Y 488.79,Z 293.602,A -85,B 0,C 180,E1 -6471.733,E2 -6471.733} C_VEL
LIN {X 0,Y 488.858,Z 293.591,A -85,B 0,C 180,E1 -6474.224,E2 -6474.224} C_VEL
LIN {X 0,Y 488.961,Z 293.578,A -85,B 0,C 180,E1 -6477.529,E2 -6477.529} C_VEL
LIN {X 0,Y 488.939,Z 293.583,A -85,B 0,C 180,E1 -6480.824,E2 -6480.824} C_VEL
LIN {X 0,Y 488.957,Z 293.581,A -85,B 0,C 180,E1 -6482.471,E2 -6482.471} C_VEL
LIN {X 0,Y 488.843,Z 293.592,A -85,B 0,C 180,E1 -6485.776,E2 -6485.776} C_VEL
LIN {X 0,Y 488.786,Z 293.601,A -85,B 0,C 180,E1 -6488.267,E2 -6488.267} C_VEL
LIN {X 0,Y 488.811,Z 293.598,A -85,B 0,C 180,E1 -6491.612,E2 -6491.612} C_VEL
LIN {X 0,Y 488.763,Z 293.604,A -85,B 0,C 180,E1 -6495,E2 -6495} C_VEL
LIN {X 0,Y 488.75,Z 293.606,A -85,B 0,C 180,E1 -6498.442,E2 -6498.442} C_VEL
LIN {X 0,Y 488.712,Z 293.609,A -85,B 0,C 180,E1 -6501.071,E2 -6501.071} C_VEL
LIN {X 0,Y 488.679,Z 293.615,A -85,B 0,C 180,E1 -6503.746,E2 -6503.746} C_VEL
LIN {X 0,Y 488.721,Z 293.609,A -85,B 0,C 180,E1 -6506.474,E2 -6506.474} C_VEL
LIN {X 0,Y 488.714,Z 293.608,A -85,B 0,C 180,E1 -6509.271,E2 -6509.271} C_VEL
LIN {X 0,Y 488.707,Z 293.611,A -85,B 0,C 180,E1 -6512.147,E2 -6512.147} C_VEL
LIN {X 0,Y 488.72,Z 293.609,A -85,B 0,C 180,E1 -6515.115,E2 -6515.115} C_VEL
LIN {X 0,Y 488.683,Z 293.614,A -85,B 0,C 180,E1 -6518.2,E2 -6518.2} C_VEL
LIN {X 0,Y 488.722,Z 293.611,A -85,B 0,C 180,E1 -6520.345,E2 -6520.345} C_VEL
LIN {X 0,Y 488.682,Z 293.614,A -85,B 0,C 180,E1 -6523.655,E2 -6523.655} C_VEL
LIN {X 0,Y 488.681,Z 293.612,A -85,B 0,C 180,E1 -6526.345,E2 -6526.345} C_VEL
LIN {X 0,Y 488.721,Z 293.61,A -85,B 0,C 180,E1 -6529.675,E2 -6529.675} C_VEL
LIN {X 0,Y 488.741,Z 293.712,A -85,B 0,C 180,E1 -6530.483,E2 -6530.483} C_VEL
LIN {X 0,Y 490.164,Z 301.502,A -85,B 0,C 180,E1 -6533.411,E2 -6533.411} C_VEL
LIN {X 0,Y 490.294,Z 306.05,A -85,B 0,C 180,E1 -6535.014,E2 -6535.014} C_VEL
LIN {X 0,Y 489.881,Z 314.765,A -85,B 0,C 180,E1 -6537.939,E2 -6537.939} C_VEL
LIN {X 0,Y 489.449,Z 324.664,A -85,B 0,C 180,E1 -6541.152,E2 -6541.152} C_VEL
LIN {X 0,Y 489.109,Z 333.759,A -85,B 0,C 180,E1 -6544.007,E2 -6544.007} C_VEL
LIN {X 0,Y 488.805,Z 343.36,A -85,B 0,C 180,E1 -6546.954,E2 -6546.954} C_VEL
LIN {X 0,Y 488.602,Z 352.871,A -85,B 0,C 180,E1 -6549.805,E2 -6549.805} C_VEL
LIN {X 0,Y 488.38,Z 363.19,A -85,B 0,C 180,E1 -6552.842,E2 -6552.842} C_VEL
LIN {X 0,Y 488.249,Z 371.692,A -85,B 0,C 180,E1 -6555.277,E2 -6555.277} C_VEL
LIN {X 0,Y 490.097,Z 385.796,A -85,B 0,C 180,E1 -6555.678,E2 -6555.678} C_VEL
LIN {X 0,Y 490.661,Z 390.421,A -85,B 0,C 180,E1 -6555.854,E2 -6555.854} C_VEL
LIN {X 0,Y 490.301,Z 402.6,A -85,B 0,C 180,E1 -6556.372,E2 -6556.372} C_VEL
LIN {X 0,Y 489.834,Z 414.872,A -85,B 0,C 180,E1 -6557.077,E2 -6557.077} C_VEL
LIN {X 0,Y 489.412,Z 425.844,A -85,B 0,C 180,E1 -6557.88,E2 -6557.88} C_VEL
LIN {X 0,Y 489.08,Z 436.114,A -85,B 0,C 180,E1 -6558.814,E2 -6558.814} C_VEL
LIN {X 0,Y 488.715,Z 445.391,A -85,B 0,C 180,E1 -6559.854,E2 -6559.854} C_VEL
LIN {X 0,Y 488.408,Z 454.427,A -85,B 0,C 180,E1 -6561.101,E2 -6561.101} C_VEL
LIN {X 0,Y 488.215,Z 461.712,A -85,B 0,C 180,E1 -6562.348,E2 -6562.348} C_VEL
LIN {X 0,Y 488.076,Z 467.113,A -85,B 0,C 180,E1 -6563.495,E2 -6563.495} C_VEL
LIN {X 0,Y 488.055,Z 471.414,A -85,B 0,C 180,E1 -6564.629,E2 -6564.629} C_VEL
LIN {X 0,Y 487.989,Z 475.064,A -85,B 0,C 180,E1 -6565.871,E2 -6565.871} C_VEL
LIN {X 0,Y 487.974,Z 476.946,A -85,B 0,C 180,E1 -6566.697,E2 -6566.697} C_VEL
LIN {X 0,Y 487.989,Z 478.36,A -85,B 0,C 180,E1 -6567.524,E2 -6567.524} C_VEL
LIN {X 0,Y 487.85,Z 479.956,A -85,B 0,C 180,E1 -6569.175,E2 -6569.175} C_VEL
LIN {X 0,Y 487.85,Z 480.164,A -85,B 0,C 180,E1 -6570,E2 -6570} C_VEL
LIN {X 0,Y 487.851,Z 479.934,A -85,B 0,C 180,E1 -6570.825,E2 -6570.825} C_VEL
LIN {X 0,Y 487.991,Z 478.286,A -85,B 0,C 180,E1 -6572.476,E2 -6572.476} C_VEL
LIN {X 0,Y 487.986,Z 476.849,A -85,B 0,C 180,E1 -6573.303,E2 -6573.303} C_VEL
LIN {X 0,Y 487.946,Z 473.836,A -85,B 0,C 180,E1 -6574.544,E2 -6574.544} C_VEL
LIN {X 0,Y 488.068,Z 469.777,A -85,B 0,C 180,E1 -6575.785,E2 -6575.785} C_VEL
LIN {X 0,Y 488.182,Z 463.532,A -85,B 0,C 180,E1 -6577.237,E2 -6577.237} C_VEL
LIN {X 0,Y 488.34,Z 456.717,A -85,B 0,C 180,E1 -6578.483,E2 -6578.483} C_VEL
LIN {X 0,Y 488.57,Z 448.274,A -85,B 0,C 180,E1 -6579.731,E2 -6579.731} C_VEL
LIN {X 0,Y 488.881,Z 439.619,A -85,B 0,C 180,E1 -6580.771,E2 -6580.771} C_VEL
LIN {X 0,Y 489.234,Z 428.968,A -85,B 0,C 180,E1 -6581.811,E2 -6581.811} C_VEL
LIN {X 0,Y 489.644,Z 417.414,A -85,B 0,C 180,E1 -6582.717,E2 -6582.717} C_VEL
LIN {X 0,Y 490.149,Z 404.921,A -85,B 0,C 180,E1 -6583.474,E2 -6583.474} C_VEL
LIN {X 0,Y 490.558,Z 392.457,A -85,B 0,C 180,E1 -6584.043,E2 -6584.043} C_VEL
LIN {X 0,Y 490.356,Z 387.779,A -85,B 0,C 180,E1 -6584.221,E2 -6584.221} C_VEL
LIN {X 0,Y 488.638,Z 374.169,A -85,B 0,C 180,E1 -6584.651,E2 -6584.651} C_VEL
LIN {X 0,Y 488.239,Z 370.684,A -85,B 0,C 180,E1 -6584.75,E2 -6584.75} C_VEL
LIN {X 0,Y 488.358,Z 360.747,A -85,B 0,C 180,E1 -6587.591,E2 -6587.591} C_VEL
LIN {X 0,Y 488.578,Z 349.791,A -85,B 0,C 180,E1 -6590.771,E2 -6590.771} C_VEL
LIN {X 0,Y 488.751,Z 339.812,A -85,B 0,C 180,E1 -6593.743,E2 -6593.743} C_VEL
LIN {X 0,Y 489.091,Z 329.083,A -85,B 0,C 180,E1 -6597.012,E2 -6597.012} C_VEL
LIN {X 0,Y 489.449,Z 318.19,A -85,B 0,C 180,E1 -6600.51,E2 -6600.51} C_VEL
LIN {X 0,Y 489.932,Z 308.749,A -85,B 0,C 180,E1 -6603.695,E2 -6603.695} C_VEL
LIN {X 0,Y 490.207,Z 302.251,A -85,B 0,C 180,E1 -6606.002,E2 -6606.002} C_VEL
LIN {X 0,Y 489.13,Z 295.685,A -85,B 0,C 180,E1 -6608.607,E2 -6608.607} C_VEL
LIN {X 0,Y 488.707,Z 293.609,A -85,B 0,C 180,E1 -6609.521,E2 -6609.521} C_VEL
LIN {X 0,Y 488.714,Z 293.613,A -85,B 0,C 180,E1 -6612.827,E2 -6612.827} C_VEL
LIN {X 0,Y 488.704,Z 293.616,A -85,B 0,C 180,E1 -6615.976,E2 -6615.976} C_VEL
LIN {X 0,Y 488.711,Z 293.613,A -85,B 0,C 180,E1 -6618.585,E2 -6618.585} C_VEL
LIN {X 0,Y 488.709,Z 293.615,A -85,B 0,C 180,E1 -6620.947,E2 -6620.947} C_VEL
LIN {X 0,Y 488.682,Z 293.615,A -85,B 0,C 180,E1 -6623.868,E2 -6623.868} C_VEL
LIN {X 0,Y 488.743,Z 293.608,A -85,B 0,C 180,E1 -6626.877,E2 -6626.877} C_VEL
LIN {X 0,Y 488.729,Z 293.609,A -85,B 0,C 180,E1 -6629.781,E2 -6629.781} C_VEL
LIN {X 0,Y 488.797,Z 293.601,A -85,B 0,C 180,E1 -6633.056,E2 -6633.056} C_VEL
LIN {X 0,Y 488.695,Z 293.614,A -85,B 0,C 180,E1 -6636.254,E2 -6636.254} C_VEL
LIN {X 0,Y 488.752,Z 293.607,A -85,B 0,C 180,E1 -6639.176,E2 -6639.176} C_VEL
LIN {X 0,Y 488.754,Z 293.605,A -85,B 0,C 180,E1 -6641.631,E2 -6641.631} C_VEL
LIN {X 0,Y 488.768,Z 293.604,A -85,B 0,C 180,E1 -6645,E2 -6645} C_VEL
LIN {X 0,Y 488.812,Z 293.598,A -85,B 0,C 180,E1 -6648.388,E2 -6648.388} C_VEL
LIN {X 0,Y 488.786,Z 293.601,A -85,B 0,C 180,E1 -6651.733,E2 -6651.733} C_VEL
LIN {X 0,Y 488.842,Z 293.596,A -85,B 0,C 180,E1 -6654.224,E2 -6654.224} C_VEL
LIN {X 0,Y 488.966,Z 293.579,A -85,B 0,C 180,E1 -6657.529,E2 -6657.529} C_VEL
LIN {X 0,Y 488.94,Z 293.582,A -85,B 0,C 180,E1 -6660.823,E2 -6660.823} C_VEL
LIN {X 0,Y 488.967,Z 293.58,A -85,B 0,C 180,E1 -6662.471,E2 -6662.471} C_VEL
LIN {X 0,Y 488.845,Z 293.595,A -85,B 0,C 180,E1 -6665.776,E2 -6665.776} C_VEL
LIN {X 0,Y 488.764,Z 293.606,A -85,B 0,C 180,E1 -6668.267,E2 -6668.267} C_VEL
LIN {X 0,Y 488.507,Z 293.639,A -85,B 0,C 180,E1 -6671.62,E2 -6671.62} C_VEL
LIN {X 0,Y 488.387,Z 294.061,A -85,B 0,C 180,E1 -6672.466,E2 -6672.466} C_VEL
LIN {X 0,Y 488.36,Z 296.861,A -85,B 0,C 180,E1 -6675.376,E2 -6675.376} C_VEL
LIN {X 0,Y 488.212,Z 299.885,A -85,B 0,C 180,E1 -6678.463,E2 -6678.463} C_VEL
LIN {X 0,Y 488.184,Z 302.445,A -85,B 0,C 180,E1 -6681.094,E2 -6681.094} C_VEL
LIN {X 0,Y 488.139,Z 304.741,A -85,B 0,C 180,E1 -6683.408,E2 -6683.408} C_VEL
LIN {X 0,Y 490.909,Z 316.161,A -85,B 0,C 180,E1 -6683.828,E2 -6683.828} C_VEL
LIN {X 0,Y 490.764,Z 329.2,A -85,B 0,C 180,E1 -6684.369,E2 -6684.369} C_VEL
LIN {X 0,Y 490.43,Z 340.684,A -85,B 0,C 180,E1 -6685.008,E2 -6685.008} C_VEL
LIN {X 0,Y 489.99,Z 352.079,A -85,B 0,C 180,E1 -6685.828,E2 -6685.828} C_VEL
LIN {X 0,Y 489.546,Z 363.149,A -85,B 0,C 180,E1 -6686.831,E2 -6686.831} C_VEL
LIN {X 0,Y 489.215,Z 372.038,A -85,B 0,C 180,E1 -6687.833,E2 -6687.833} C_VEL
LIN {X 0,Y 488.916,Z 380.219,A -85,B 0,C 180,E1 -6688.963,E2 -6688.963} C_VEL
LIN {X 0,Y 488.568,Z 388.206,A -85,B 0,C 180,E1 -6690.333,E2 -6690.333} C_VEL
LIN {X 0,Y 488.377,Z 393.776,A -85,B 0,C 180,E1 -6691.539,E2 -6691.539} C_VEL
LIN {X 0,Y 488.216,Z 397.946,A -85,B 0,C 180,E1 -6692.672,E2 -6692.672} C_VEL
LIN {X 0,Y 488.093,Z 402.098,A -85,B 0,C 180,E1 -6694.163,E2 -6694.163} C_VEL
LIN {X 0,Y 487.952,Z 404.078,A -85,B 0,C 180,E1 -6695.178,E2 -6695.178} C_VEL
LIN {X 0,Y 487.93,Z 405.493,A -85,B 0,C 180,E1 -6696.233,E2 -6696.233} C_VEL
LIN {X 0,Y 487.86,Z 406.355,A -85,B 0,C 180,E1 -6697.597,E2 -6697.597} C_VEL
LIN {X 0,Y 487.89,Z 406.157,A -85,B 0,C 180,E1 -6698.934,E2 -6698.934} C_VEL
LIN {X 0,Y 487.947,Z 404.747,A -85,B 0,C 180,E1 -6700.402,E2 -6700.402} C_VEL
LIN {X 0,Y 488.116,Z 401.706,A -85,B 0,C 180,E1 -6702.029,E2 -6702.029} C_VEL
LIN {X 0,Y 488.207,Z 398.476,A -85,B 0,C 180,E1 -6703.196,E2 -6703.196} C_VEL
LIN {X 0,Y 488.318,Z 394.254,A -85,B 0,C 180,E1 -6704.372,E2 -6704.372} C_VEL
LIN {X 0,Y 488.509,Z 387.848,A -85,B 0,C 180,E1 -6705.769,E2 -6705.769} C_VEL
LIN {X 0,Y 488.854,Z 379.681,A -85,B 0,C 180,E1 -6707.155,E2 -6707.155} C_VEL
LIN {X 0,Y 489.165,Z 370.961,A -85,B 0,C 180,E1 -6708.34,E2 -6708.34} C_VEL
LIN {X 0,Y 489.541,Z 361.583,A -85,B 0,C 180,E1 -6709.367,E2 -6709.367} C_VEL
LIN {X 0,Y 489.947,Z 351.087,A -85,B 0,C 180,E1 -6710.301,E2 -6710.301} C_VEL
LIN {X 0,Y 490.37,Z 339.497,A -85,B 0,C 180,E1 -6711.122,E2 -6711.122} C_VEL
LIN {X 0,Y 490.725,Z 327.947,A -85,B 0,C 180,E1 -6711.753,E2 -6711.753} C_VEL
LIN {X 0,Y 490.872,Z 316.149,A -85,B 0,C 180,E1 -6712.24,E2 -6712.24} C_VEL
LIN {X 0,Y 490.086,Z 312.245,A -85,B 0,C 180,E1 -6712.395,E2 -6712.395} C_VEL
LIN {X 0,Y 489.006,Z 309.094,A -85,B 0,C 180,E1 -6712.597,E2 -6712.597} C_VEL
LIN {X 0,Y 487.617,Z 306.679,A -85,B 0,C 180,E1 -6712.9,E2 -6712.9} C_VEL
LIN {X 0,Y 485.362,Z 304.221,A -85,B 0,C 180,E1 -6713.47,E2 -6713.47} C_VEL
LIN {X 0,Y 483.234,Z 302.853,A -85,B 0,C 180,E1 -6714.143,E2 -6714.143} C_VEL
LIN {X 0,Y 481.264,Z 301.836,A -85,B 0,C 180,E1 -6715.119,E2 -6715.119} C_VEL
LIN {X 0,Y 480.966,Z 301.334,A -85,B 0,C 180,E1 -6715.621,E2 -6715.621} C_VEL
LIN {X 0,Y 481.032,Z 298.558,A -85,B 0,C 180,E1 -6718.266,E2 -6718.266} C_VEL
LIN {X 0,Y 481.087,Z 295.461,A -85,B 0,C 180,E1 -6721.225,E2 -6721.225} C_VEL
LIN {X 0,Y 481.105,Z 294.563,A -85,B 0,C 180,E1 -6722.13,E2 -6722.13} C_VEL
LIN {X 0,Y 481.421,Z 294.521,A -85,B 0,C 180,E1 -6724.953,E2 -6724.953} C_VEL
LIN {X 0,Y 481.644,Z 294.49,A -85,B 0,C 180,E1 -6727.704,E2 -6727.704} C_VEL
LIN {X 0,Y 481.704,Z 294.481,A -85,B 0,C 180,E1 -6730.393,E2 -6730.393} C_VEL
LIN {X 0,Y 481.678,Z 294.486,A -85,B 0,C 180,E1 -6733.033,E2 -6733.033} C_VEL
LIN {X 0,Y 481.69,Z 294.485,A -85,B 0,C 180,E1 -6735.639,E2 -6735.639} C_VEL
LIN {X 0,Y 481.752,Z 294.475,A -85,B 0,C 180,E1 -6738.215,E2 -6738.215} C_VEL
LIN {X 0,Y 481.763,Z 294.475,A -85,B 0,C 180,E1 -6741.612,E2 -6741.612} C_VEL
LIN {X 0,Y 481.779,Z 294.475,A -85,B 0,C 180,E1 -6744.979,E2 -6744.979} C_VEL
LIN {X 0,Y 481.929,Z 294.455,A -85,B 0,C 180,E1 -6747.493,E2 -6747.493} C_VEL
LIN {X 0,Y 481.943,Z 294.451,A -85,B 0,C 180,E1 -6750,E2 -6750} C_VEL
LIN {X 0,Y 481.93,Z 294.455,A -85,B 0,C 180,E1 -6752.507,E2 -6752.507} C_VEL
LIN {X 0,Y 481.798,Z 294.472,A -85,B 0,C 180,E1 -6755.861,E2 -6755.861} C_VEL
LIN {X 0,Y 481.763,Z 294.477,A -85,B 0,C 180,E1 -6758.388,E2 -6758.388} C_VEL
LIN {X 0,Y 481.752,Z 294.475,A -85,B 0,C 180,E1 -6761.785,E2 -6761.785} C_VEL
LIN {X 0,Y 481.743,Z 294.477,A -85,B 0,C 180,E1 -6765.224,E2 -6765.224} C_VEL
LIN {X 0,Y 481.708,Z 294.484,A -85,B 0,C 180,E1 -6768.722,E2 -6768.722} C_VEL
LIN {X 0,Y 481.648,Z 294.49,A -85,B 0,C 180,E1 -6771.395,E2 -6771.395} C_VEL
LIN {X 0,Y 481.679,Z 294.488,A -85,B 0,C 180,E1 -6774.113,E2 -6774.113} C_VEL
LIN {X 0,Y 481.747,Z 294.477,A -85,B 0,C 180,E1 -6777.139,E2 -6777.139} C_VEL
LIN {X 0,Y 481.679,Z 294.487,A -85,B 0,C 180,E1 -6779.741,E2 -6779.741} C_VEL
LIN {X 0,Y 481.672,Z 294.486,A -85,B 0,C 180,E1 -6782.675,E2 -6782.675} C_VEL
LIN {X 0,Y 481.638,Z 294.491,A -85,B 0,C 180,E1 -6785.71,E2 -6785.71} C_VEL
LIN {X 0,Y 481.673,Z 294.486,A -85,B 0,C 180,E1 -6788.859,E2 -6788.859} C_VEL
LIN {X 0,Y 481.655,Z 294.489,A -85,B 0,C 180,E1 -6791.913,E2 -6791.913} C_VEL
LIN {X 0,Y 481.657,Z 294.488,A -85,B 0,C 180,E1 -6794.458,E2 -6794.458} C_VEL
LIN {X 0,Y 481.65,Z 294.492,A -85,B 0,C 180,E1 -6797.84,E2 -6797.84} C_VEL
LIN {X 0,Y 481.684,Z 294.485,A -85,B 0,C 180,E1 -6800.651,E2 -6800.651} C_VEL
LIN {X 0,Y 481.63,Z 294.493,A -85,B 0,C 180,E1 -6803.376,E2 -6803.376} C_VEL
LIN {X 0,Y 481.68,Z 294.485,A -85,B 0,C 180,E1 -6806.328,E2 -6806.328} C_VEL
LIN {X 0,Y 481.654,Z 294.49,A -85,B 0,C 180,E1 -6809.418,E2 -6809.418} C_VEL
LIN {X 0,Y 481.695,Z 294.485,A -85,B 0,C 180,E1 -6812.168,E2 -6812.168} C_VEL
LIN {X 0,Y 481.682,Z 294.487,A -85,B 0,C 180,E1 -6814.968,E2 -6814.968} C_VEL
LIN {X 0,Y 481.653,Z 294.49,A -85,B 0,C 180,E1 -6817.705,E2 -6817.705} C_VEL
LIN {X 0,Y 481.709,Z 294.482,A -85,B 0,C 180,E1 -6820.393,E2 -6820.393} C_VEL
LIN {X 0,Y 481.682,Z 294.487,A -85,B 0,C 180,E1 -6823.034,E2 -6823.034} C_VEL
LIN {X 0,Y 481.693,Z 294.484,A -85,B 0,C 180,E1 -6825.639,E2 -6825.639} C_VEL
LIN {X 0,Y 481.756,Z 294.477,A -85,B 0,C 180,E1 -6828.215,E2 -6828.215} C_VEL
LIN {X 0,Y 481.744,Z 294.479,A -85,B 0,C 180,E1 -6831.611,E2 -6831.611} C_VEL
LIN {X 0,Y 481.819,Z 294.467,A -85,B 0,C 180,E1 -6834.14,E2 -6834.14} C_VEL
LIN {X 0,Y 481.927,Z 294.454,A -85,B 0,C 180,E1 -6837.493,E2 -6837.493} C_VEL
LIN {X 0,Y 481.891,Z 294.461,A -85,B 0,C 180,E1 -6840.836,E2 -6840.836} C_VEL
LIN {X 0,Y 481.923,Z 294.458,A -85,B 0,C 180,E1 -6842.508,E2 -6842.508} C_VEL
LIN {X 0,Y 481.801,Z 294.469,A -85,B 0,C 180,E1 -6845.861,E2 -6845.861} C_VEL
LIN {X 0,Y 481.742,Z 294.478,A -85,B 0,C 180,E1 -6848.389,E2 -6848.389} C_VEL
LIN {X 0,Y 481.756,Z 294.477,A -85,B 0,C 180,E1 -6851.785,E2 -6851.785} C_VEL
LIN {X 0,Y 481.745,Z 294.479,A -85,B 0,C 180,E1 -6855.224,E2 -6855.224} C_VEL
LIN {X 0,Y 481.712,Z 294.482,A -85,B 0,C 180,E1 -6858.722,E2 -6858.722} C_VEL
LIN {X 0,Y 481.65,Z 294.487,A -85,B 0,C 180,E1 -6861.395,E2 -6861.395} C_VEL
LIN {X 0,Y 481.661,Z 294.488,A -85,B 0,C 180,E1 -6864.114,E2 -6864.114} C_VEL
LIN {X 0,Y 481.698,Z 294.484,A -85,B 0,C 180,E1 -6867.127,E2 -6867.127} C_VEL
LIN {X 0,Y 481.677,Z 294.486,A -85,B 0,C 180,E1 -6869.741,E2 -6869.741} C_VEL
LIN {X 0,Y 481.676,Z 294.487,A -85,B 0,C 180,E1 -6872.674,E2 -6872.674} C_VEL
LIN {X 0,Y 481.64,Z 294.491,A -85,B 0,C 180,E1 -6875.709,E2 -6875.709} C_VEL
LIN {X 0,Y 481.674,Z 294.487,A -85,B 0,C 180,E1 -6878.859,E2 -6878.859} C_VEL
LIN {X 0,Y 481.65,Z 294.492,A -85,B 0,C 180,E1 -6881.912,E2 -6881.912} C_VEL
LIN {X 0,Y 481.657,Z 294.49,A -85,B 0,C 180,E1 -6884.458,E2 -6884.458} C_VEL
LIN {X 0,Y 481.646,Z 294.489,A -85,B 0,C 180,E1 -6887.839,E2 -6887.839} C_VEL
LIN {X 0,Y 481.722,Z 294.587,A -85,B 0,C 180,E1 -6890.224,E2 -6890.224} C_VEL
LIN {X 0,Y 483.208,Z 302.869,A -85,B 0,C 180,E1 -6893.393,E2 -6893.393} C_VEL
LIN {X 0,Y 483.328,Z 307.317,A -85,B 0,C 180,E1 -6894.98,E2 -6894.98} C_VEL
LIN {X 0,Y 482.875,Z 316.126,A -85,B 0,C 180,E1 -6897.987,E2 -6897.987} C_VEL
LIN {X 0,Y 482.406,Z 326.085,A -85,B 0,C 180,E1 -6901.264,E2 -6901.264} C_VEL
LIN {X 0,Y 482.063,Z 334.849,A -85,B 0,C 180,E1 -6904.064,E2 -6904.064} C_VEL
LIN {X 0,Y 481.706,Z 345.123,A -85,B 0,C 180,E1 -6907.255,E2 -6907.255} C_VEL
LIN {X 0,Y 481.463,Z 355.398,A -85,B 0,C 180,E1 -6910.383,E2 -6910.383} C_VEL
LIN {X 0,Y 481.278,Z 364.202,A -85,B 0,C 180,E1 -6913.019,E2 -6913.019} C_VEL
LIN {X 0,Y 481.183,Z 371.113,A -85,B 0,C 180,E1 -6915.056,E2 -6915.056} C_VEL
LIN {X 0,Y 482.995,Z 385.168,A -85,B 0,C 180,E1 -6915.463,E2 -6915.463} C_VEL
LIN {X 0,Y 483.719,Z 391.287,A -85,B 0,C 180,E1 -6915.7,E2 -6915.7} C_VEL
LIN {X 0,Y 483.343,Z 403.02,A -85,B 0,C 180,E1 -6916.226,E2 -6916.226} C_VEL
LIN {X 0,Y 482.8,Z 416.044,A -85,B 0,C 180,E1 -6917.003,E2 -6917.003} C_VEL
LIN {X 0,Y 482.353,Z 427.086,A -85,B 0,C 180,E1 -6917.852,E2 -6917.852} C_VEL
LIN {X 0,Y 481.97,Z 437.542,A -85,B 0,C 180,E1 -6918.86,E2 -6918.86} C_VEL
LIN {X 0,Y 481.577,Z 446.486,A -85,B 0,C 180,E1 -6919.914,E2 -6919.914} C_VEL
LIN {X 0,Y 481.29,Z 455.234,A -85,B 0,C 180,E1 -6921.18,E2 -6921.18} C_VEL
LIN {X 0,Y 481.104,Z 462.22,A -85,B 0,C 180,E1 -6922.445,E2 -6922.445} C_VEL
LIN {X 0,Y 480.936,Z 468.223,A -85,B 0,C 180,E1 -6923.813,E2 -6923.813} C_VEL
LIN {X 0,Y 480.906,Z 472.211,A -85,B 0,C 180,E1 -6924.97,E2 -6924.97} C_VEL
LIN {X 0,Y 480.887,Z 474.532,A -85,B 0,C 180,E1 -6925.809,E2 -6925.809} C_VEL
LIN {X 0,Y 480.901,Z 476.417,A -85,B 0,C 180,E1 -6926.649,E2 -6926.649} C_VEL
LIN {X 0,Y 480.926,Z 477.831,A -85,B 0,C 180,E1 -6927.487,E2 -6927.487} C_VEL
LIN {X 0,Y 480.775,Z 479.423,A -85,B 0,C 180,E1 -6929.162,E2 -6929.162} C_VEL
LIN {X 0,Y 480.772,Z 479.629,A -85,B 0,C 180,E1 -6930,E2 -6930} C_VEL
LIN {X 0,Y 480.776,Z 479.397,A -85,B 0,C 180,E1 -6930.838,E2 -6930.838} C_VEL
LIN {X 0,Y 480.928,Z 477.742,A -85,B 0,C 180,E1 -6932.513,E2 -6932.513} C_VEL
LIN {X 0,Y 480.913,Z 476.301,A -85,B 0,C 180,E1 -6933.351,E2 -6933.351} C_VEL
LIN {X 0,Y 480.861,Z 473.279,A -85,B 0,C 180,E1 -6934.611,E2 -6934.611} C_VEL
LIN {X 0,Y 480.964,Z 469.209,A -85,B 0,C 180,E1 -6935.871,E2 -6935.871} C_VEL
LIN {X 0,Y 481.107,Z 462.951,A -85,B 0,C 180,E1 -6937.344,E2 -6937.344} C_VEL
LIN {X 0,Y 481.278,Z 456.127,A -85,B 0,C 180,E1 -6938.608,E2 -6938.608} C_VEL
LIN {X 0,Y 481.501,Z 447.673,A -85,B 0,C 180,E1 -6939.875,E2 -6939.875} C_VEL
LIN {X 0,Y 481.857,Z 439.009,A -85,B 0,C 180,E1 -6940.93,E2 -6940.93} C_VEL
LIN {X 0,Y 482.236,Z 428.606,A -85,B 0,C 180,E1 -6941.962,E2 -6941.962} C_VEL
LIN {X 0,Y 482.645,Z 417.796,A -85,B 0,C 180,E1 -6942.83,E2 -6942.83} C_VEL
LIN {X 0,Y 483.142,Z 406.265,A -85,B 0,C 180,E1 -6943.566,E2 -6943.566} C_VEL
LIN {X 0,Y 483.557,Z 394.405,A -85,B 0,C 180,E1 -6944.144,E2 -6944.144} C_VEL
LIN {X 0,Y 483.417,Z 388.662,A -85,B 0,C 180,E1 -6944.376,E2 -6944.376} C_VEL
LIN {X 0,Y 481.733,Z 374.918,A -85,B 0,C 180,E1 -6944.835,E2 -6944.835} C_VEL
LIN {X 0,Y 481.172,Z 370.109,A -85,B 0,C 180,E1 -6944.972,E2 -6944.972} C_VEL
LIN {X 0,Y 481.288,Z 360.2,A -85,B 0,C 180,E1 -6947.858,E2 -6947.858} C_VEL
LIN {X 0,Y 481.515,Z 349.894,A -85,B 0,C 180,E1 -6950.913,E2 -6950.913} C_VEL
LIN {X 0,Y 481.702,Z 339.324,A -85,B 0,C 180,E1 -6954.112,E2 -6954.112} C_VEL
LIN {X 0,Y 482.057,Z 329.435,A -85,B 0,C 180,E1 -6957.21,E2 -6957.21} C_VEL
LIN {X 0,Y 482.387,Z 320.339,A -85,B 0,C 180,E1 -6960.175,E2 -6960.175} C_VEL
LIN {X 0,Y 482.836,Z 311.785,A -85,B 0,C 180,E1 -6963.082,E2 -6963.082} C_VEL
LIN {X 0,Y 483.244,Z 304.824,A -85,B 0,C 180,E1 -6965.573,E2 -6965.573} C_VEL
LIN {X 0,Y 482.803,Z 300.574,A -85,B 0,C 180,E1 -6967.223,E2 -6967.223} C_VEL
LIN {X 0,Y 481.692,Z 294.484,A -85,B 0,C 180,E1 -6969.776,E2 -6969.776} C_VEL
LIN {X 0,Y 481.648,Z 294.493,A -85,B 0,C 180,E1 -6973.149,E2 -6973.149} C_VEL
LIN {X 0,Y 481.662,Z 294.493,A -85,B 0,C 180,E1 -6975.641,E2 -6975.641} C_VEL
LIN {X 0,Y 481.66,Z 294.493,A -85,B 0,C 180,E1 -6978.958,E2 -6978.958} C_VEL
LIN {X 0,Y 481.66,Z 294.491,A -85,B 0,C 180,E1 -6981.993,E2 -6981.993} C_VEL
LIN {X 0,Y 481.693,Z 294.485,A -85,B 0,C 180,E1 -6985.318,E2 -6985.318} C_VEL
LIN {X 0,Y 481.65,Z 294.491,A -85,B 0,C 180,E1 -6988.312,E2 -6988.312} C_VEL
LIN {X 0,Y 481.706,Z 294.484,A -85,B 0,C 180,E1 -6991.219,E2 -6991.219} C_VEL
LIN {X 0,Y 481.706,Z 294.485,A -85,B 0,C 180,E1 -6994.043,E2 -6994.043} C_VEL
LIN {X 0,Y 481.679,Z 294.487,A -85,B 0,C 180,E1 -6996.812,E2 -6996.812} C_VEL
LIN {X 0,Y 481.701,Z 294.483,A -85,B 0,C 180,E1 -6999.503,E2 -6999.503} C_VEL
LIN {X 0,Y 481.698,Z 294.484,A -85,B 0,C 180,E1 -7002.158,E2 -7002.158} C_VEL
LIN {X 0,Y 481.748,Z 294.477,A -85,B 0,C 180,E1 -7004.776,E2 -7004.776} C_VEL
LIN {X 0,Y 481.757,Z 294.478,A -85,B 0,C 180,E1 -7008.215,E2 -7008.215} C_VEL
LIN {X 0,Y 481.742,Z 294.478,A -85,B 0,C 180,E1 -7011.611,E2 -7011.611} C_VEL
LIN {X 0,Y 481.801,Z 294.473,A -85,B 0,C 180,E1 -7014.139,E2 -7014.139} C_VEL
LIN {X 0,Y 481.933,Z 294.455,A -85,B 0,C 180,E1 -7017.492,E2 -7017.492} C_VEL
LIN {X 0,Y 481.892,Z 294.46,A -85,B 0,C 180,E1 -7020.836,E2 -7020.836} C_VEL
LIN {X 0,Y 481.934,Z 294.456,A -85,B 0,C 180,E1 -7022.507,E2 -7022.507} C_VEL
LIN {X 0,Y 481.804,Z 294.472,A -85,B 0,C 180,E1 -7025.86,E2 -7025.86} C_VEL
LIN {X 0,Y 481.715,Z 294.484,A -85,B 0,C 180,E1 -7028.389,E2 -7028.389} C_VEL
LIN {X 0,Y 481.44,Z 294.519,A -85,B 0,C 180,E1 -7031.793,E2 -7031.793} C_VEL
LIN {X 0,Y 481.311,Z 297.548,A -85,B 0,C 180,E1 -7035.238,E2 -7035.238} C_VEL
LIN {X 0,Y 481.137,Z 300.972,A -85,B 0,C 180,E1 -7038.745,E2 -7038.745} C_VEL
LIN {X 0,Y 481.116,Z 303.571,A -85,B 0,C 180,E1 -7041.419,E2 -7041.419} C_VEL
LIN {X 0,Y 481.07,Z 305.292,A -85,B 0,C 180,E1 -7043.175,E2 -7043.175} C_VEL
LIN {X 0,Y 484.146,Z 317.743,A -85,B 0,C 180,E1 -7043.66,E2 -7043.66} C_VEL
LIN {X 0,Y 483.887,Z 330.864,A -85,B 0,C 180,E1 -7044.224,E2 -7044.224} C_VEL
LIN {X 0,Y 483.461,Z 342.959,A -85,B 0,C 180,E1 -7044.934,E2 -7044.934} C_VEL
LIN {X 0,Y 482.992,Z 354.152,A -85,B 0,C 180,E1 -7045.776,E2 -7045.776} C_VEL
LIN {X 0,Y 482.599,Z 364.197,A -85,B 0,C 180,E1 -7046.72,E2 -7046.72} C_VEL
LIN {X 0,Y 482.23,Z 373.454,A -85,B 0,C 180,E1 -7047.799,E2 -7047.799} C_VEL
LIN {X 0,Y 481.853,Z 382.371,A -85,B 0,C 180,E1 -7049.084,E2 -7049.084} C_VEL
LIN {X 0,Y 481.536,Z 389.393,A -85,B 0,C 180,E1 -7050.345,E2 -7050.345} C_VEL
LIN {X 0,Y 481.29,Z 395.382,A -85,B 0,C 180,E1 -7051.714,E2 -7051.714} C_VEL
LIN {X 0,Y 481.098,Z 400.226,A -85,B 0,C 180,E1 -7053.165,E2 -7053.165} C_VEL
LIN {X 0,Y 480.942,Z 403.956,A -85,B 0,C 180,E1 -7054.744,E2 -7054.744} C_VEL
LIN {X 0,Y 480.845,Z 405.544,A -85,B 0,C 180,E1 -7055.777,E2 -7055.777} C_VEL
LIN {X 0,Y 480.807,Z 406.555,A -85,B 0,C 180,E1 -7056.82,E2 -7056.82} C_VEL
LIN {X 0,Y 480.792,Z 406.937,A -85,B 0,C 180,E1 -7057.875,E2 -7057.875} C_VEL
LIN {X 0,Y 480.839,Z 406.522,A -85,B 0,C 180,E1 -7059.226,E2 -7059.226} C_VEL
LIN {X 0,Y 480.891,Z 405.133,A -85,B 0,C 180,E1 -7060.539,E2 -7060.539} C_VEL
LIN {X 0,Y 481.053,Z 401.878,A -85,B 0,C 180,E1 -7062.225,E2 -7062.225} C_VEL
LIN {X 0,Y 481.207,Z 397.13,A -85,B 0,C 180,E1 -7063.829,E2 -7063.829} C_VEL
LIN {X 0,Y 481.392,Z 391.364,A -85,B 0,C 180,E1 -7065.259,E2 -7065.259} C_VEL
LIN {X 0,Y 481.665,Z 383.807,A -85,B 0,C 180,E1 -7066.703,E2 -7066.703} C_VEL
LIN {X 0,Y 482.025,Z 376.097,A -85,B 0,C 180,E1 -7067.879,E2 -7067.879} C_VEL
LIN {X 0,Y 482.409,Z 366.738,A -85,B 0,C 180,E1 -7069.036,E2 -7069.036} C_VEL
LIN {X 0,Y 482.825,Z 356.704,A -85,B 0,C 180,E1 -7070.037,E2 -7070.037} C_VEL
LIN {X 0,Y 483.27,Z 345.214,A -85,B 0,C 180,E1 -7070.959,E2 -7070.959} C_VEL
LIN {X 0,Y 483.707,Z 333.549,A -85,B 0,C 180,E1 -7071.683,E2 -7071.683} C_VEL
LIN {X 0,Y 484.074,Z 320.493,A -85,B 0,C 180,E1 -7072.295,E2 -7072.295} C_VEL
LIN {X 0,Y 483.822,Z 316.03,A -85,B 0,C 180,E1 -7072.469,E2 -7072.469} C_VEL
LIN {X 0,Y 480.959,Z 304.197,A -85,B 0,C 180,E1 -7072.932,E2 -7072.932} C_VEL
LIN {X 0,Y 480.966,Z 301.334,A -85,B 0,C 180,E1 -7075.621,E2 -7075.621} C_VEL
LIN {X 0,Y 480.299,Z 300.67,A -85,B 0,C 180,E1 -7076.315,E2 -7076.315} C_VEL
LIN {X 0,Y 477.435,Z 299.774,A -85,B 0,C 180,E1 -7077.446,E2 -7077.446} C_VEL
LIN {X 0,Y 475.034,Z 299.056,A -85,B 0,C 180,E1 -7078.357,E2 -7078.357} C_VEL
LIN {X 0,Y 474.037,Z 298.418,A -85,B 0,C 180,E1 -7079.06,E2 -7079.06} C_VEL
LIN {X 0,Y 473.974,Z 298.172,A -85,B 0,C 180,E1 -7079.297,E2 -7079.297} C_VEL
LIN {X 0,Y 474.014,Z 295.69,A -85,B 0,C 180,E1 -7081.676,E2 -7081.676} C_VEL
LIN {X 0,Y 474.235,Z 295.416,A -85,B 0,C 180,E1 -7083.603,E2 -7083.603} C_VEL
LIN {X 0,Y 474.544,Z 295.376,A -85,B 0,C 180,E1 -7086.667,E2 -7086.667} C_VEL
LIN {X 0,Y 474.672,Z 295.36,A -85,B 0,C 180,E1 -7089.185,E2 -7089.185} C_VEL
LIN {X 0,Y 474.646,Z 295.363,A -85,B 0,C 180,E1 -7091.884,E2 -7091.884} C_VEL
LIN {X 0,Y 474.701,Z 295.354,A -85,B 0,C 180,E1 -7094.544,E2 -7094.544} C_VEL
LIN {X 0,Y 474.706,Z 295.353,A -85,B 0,C 180,E1 -7098.037,E2 -7098.037} C_VEL
LIN {X 0,Y 474.728,Z 295.352,A -85,B 0,C 180,E1 -7101.486,E2 -7101.486} C_VEL
LIN {X 0,Y 474.749,Z 295.35,A -85,B 0,C 180,E1 -7104.904,E2 -7104.904} C_VEL
LIN {X 0,Y 474.895,Z 295.331,A -85,B 0,C 180,E1 -7107.455,E2 -7107.455} C_VEL
LIN {X 0,Y 474.914,Z 295.327,A -85,B 0,C 180,E1 -7110,E2 -7110} C_VEL
LIN {X 0,Y 474.896,Z 295.331,A -85,B 0,C 180,E1 -7112.545,E2 -7112.545} C_VEL
LIN {X 0,Y 474.759,Z 295.349,A -85,B 0,C 180,E1 -7115.948,E2 -7115.948} C_VEL
LIN {X 0,Y 474.728,Z 295.354,A -85,B 0,C 180,E1 -7118.514,E2 -7118.514} C_VEL
LIN {X 0,Y 474.706,Z 295.354,A -85,B 0,C 180,E1 -7121.962,E2 -7121.962} C_VEL
LIN {X 0,Y 474.7,Z 295.354,A -85,B 0,C 180,E1 -7125.456,E2 -7125.456} C_VEL
LIN {X 0,Y 474.663,Z 295.36,A -85,B 0,C 180,E1 -7129.01,E2 -7129.01} C_VEL
LIN {X 0,Y 474.591,Z 295.37,A -85,B 0,C 180,E1 -7131.729,E2 -7131.729} C_VEL
LIN {X 0,Y 474.661,Z 295.361,A -85,B 0,C 180,E1 -7134.493,E2 -7134.493} C_VEL
LIN {X 0,Y 474.682,Z 295.357,A -85,B 0,C 180,E1 -7137.334,E2 -7137.334} C_VEL
LIN {X 0,Y 474.604,Z 295.367,A -85,B 0,C 180,E1 -7140.81,E2 -7140.81} C_VEL
LIN {X 0,Y 474.627,Z 295.364,A -85,B 0,C 180,E1 -7143.222,E2 -7143.222} C_VEL
LIN {X 0,Y 474.59,Z 295.369,A -85,B 0,C 180,E1 -7146.324,E2 -7146.324} C_VEL
LIN {X 0,Y 474.63,Z 295.364,A -85,B 0,C 180,E1 -7149.648,E2 -7149.648} C_VEL
LIN {X 0,Y 474.608,Z 295.366,A -85,B 0,C 180,E1 -7152.935,E2 -7152.935} C_VEL
LIN {X 0,Y 474.608,Z 295.367,A -85,B 0,C 180,E1 -7155.895,E2 -7155.895} C_VEL
LIN {X 0,Y 474.631,Z 295.364,A -85,B 0,C 180,E1 -7159.041,E2 -7159.041} C_VEL
LIN {X 0,Y 474.613,Z 295.369,A -85,B 0,C 180,E1 -7161.704,E2 -7161.704} C_VEL
LIN {X 0,Y 474.626,Z 295.364,A -85,B 0,C 180,E1 -7164.726,E2 -7164.726} C_VEL
LIN {X 0,Y 474.638,Z 295.363,A -85,B 0,C 180,E1 -7167.788,E2 -7167.788} C_VEL
LIN {X 0,Y 474.626,Z 295.365,A -85,B 0,C 180,E1 -7170.885,E2 -7170.885} C_VEL
LIN {X 0,Y 474.632,Z 295.365,A -85,B 0,C 180,E1 -7173.627,E2 -7173.627} C_VEL
LIN {X 0,Y 474.638,Z 295.363,A -85,B 0,C 180,E1 -7176.642,E2 -7176.642} C_VEL
LIN {X 0,Y 474.659,Z 295.361,A -85,B 0,C 180,E1 -7180.09,E2 -7180.09} C_VEL
LIN {X 0,Y 474.642,Z 295.364,A -85,B 0,C 180,E1 -7182.774,E2 -7182.774} C_VEL
LIN {X 0,Y 474.652,Z 295.363,A -85,B 0,C 180,E1 -7185.421,E2 -7185.421} C_VEL
LIN {X 0,Y 474.709,Z 295.354,A -85,B 0,C 180,E1 -7188.038,E2 -7188.038} C_VEL
LIN {X 0,Y 474.716,Z 295.354,A -85,B 0,C 180,E1 -7191.486,E2 -7191.486} C_VEL
LIN {X 0,Y 474.782,Z 295.343,A -85,B 0,C 180,E1 -7194.053,E2 -7194.053} C_VEL
LIN {X 0,Y 474.892,Z 295.331,A -85,B 0,C 180,E1 -7197.455,E2 -7197.455} C_VEL
LIN {X 0,Y 474.916,Z 295.329,A -85,B 0,C 180,E1 -7200,E2 -7200} C_VEL
LIN {X 0,Y 474.888,Z 295.334,A -85,B 0,C 180,E1 -7202.545,E2 -7202.545} C_VEL
LIN {X 0,Y 474.761,Z 295.346,A -85,B 0,C 180,E1 -7205.948,E2 -7205.948} C_VEL
LIN {X 0,Y 474.714,Z 295.354,A -85,B 0,C 180,E1 -7208.514,E2 -7208.514} C_VEL
LIN {X 0,Y 474.71,Z 295.355,A -85,B 0,C 180,E1 -7211.962,E2 -7211.962} C_VEL
LIN {X 0,Y 474.704,Z 295.355,A -85,B 0,C 180,E1 -7215.456,E2 -7215.456} C_VEL
LIN {X 0,Y 474.667,Z 295.36,A -85,B 0,C 180,E1 -7219.01,E2 -7219.01} C_VEL
LIN {X 0,Y 474.593,Z 295.367,A -85,B 0,C 180,E1 -7221.729,E2 -7221.729} C_VEL
LIN {X 0,Y 474.64,Z 295.364,A -85,B 0,C 180,E1 -7224.494,E2 -7224.494} C_VEL
LIN {X 0,Y 474.641,Z 295.363,A -85,B 0,C 180,E1 -7227.324,E2 -7227.324} C_VEL
LIN {X 0,Y 474.606,Z 295.368,A -85,B 0,C 180,E1 -7230.23,E2 -7230.23} C_VEL
LIN {X 0,Y 474.647,Z 295.36,A -85,B 0,C 180,E1 -7233.22,E2 -7233.22} C_VEL
LIN {X 0,Y 474.592,Z 295.371,A -85,B 0,C 180,E1 -7236.323,E2 -7236.323} C_VEL
LIN {X 0,Y 474.617,Z 295.366,A -85,B 0,C 180,E1 -7239.645,E2 -7239.645} C_VEL
LIN {X 0,Y 474.604,Z 295.367,A -85,B 0,C 180,E1 -7242.233,E2 -7242.233} C_VEL
LIN {X 0,Y 474.62,Z 295.364,A -85,B 0,C 180,E1 -7245.298,E2 -7245.298} C_VEL
LIN {X 0,Y 474.618,Z 295.366,A -85,B 0,C 180,E1 -7248.214,E2 -7248.214} C_VEL
LIN {X 0,Y 474.656,Z 295.408,A -85,B 0,C 180,E1 -7249.942,E2 -7249.942} C_VEL
LIN {X 0,Y 476.252,Z 304.181,A -85,B 0,C 180,E1 -7253.355,E2 -7253.355} C_VEL
LIN {X 0,Y 476.359,Z 308.357,A -85,B 0,C 180,E1 -7254.873,E2 -7254.873} C_VEL
LIN {X 0,Y 475.901,Z 317.033,A -85,B 0,C 180,E1 -7257.883,E2 -7257.883} C_VEL
LIN {X 0,Y 475.389,Z 327.211,A -85,B 0,C 180,E1 -7261.284,E2 -7261.284} C_VEL
LIN {X 0,Y 474.967,Z 337.396,A -85,B 0,C 180,E1 -7264.589,E2 -7264.589} C_VEL
LIN {X 0,Y 474.582,Z 347.635,A -85,B 0,C 180,E1 -7267.813,E2 -7267.813} C_VEL
LIN {X 0,Y 474.362,Z 356.426,A -85,B 0,C 180,E1 -7270.527,E2 -7270.527} C_VEL
LIN {X 0,Y 474.187,Z 366.689,A -85,B 0,C 180,E1 -7273.644,E2 -7273.644} C_VEL
LIN {X 0,Y 474.103,Z 370.622,A -85,B 0,C 180,E1 -7274.827,E2 -7274.827} C_VEL
LIN {X 0,Y 475.96,Z 384.954,A -85,B 0,C 180,E1 -7275.257,E2 -7275.257} C_VEL
LIN {X 0,Y 476.783,Z 391.977,A -85,B 0,C 180,E1 -7275.542,E2 -7275.542} C_VEL
LIN {X 0,Y 476.339,Z 404.401,A -85,B 0,C 180,E1 -7276.128,E2 -7276.128} C_VEL
LIN {X 0,Y 475.814,Z 416.401,A -85,B 0,C 180,E1 -7276.874,E2 -7276.874} C_VEL
LIN {X 0,Y 475.347,Z 427.024,A -85,B 0,C 180,E1 -7277.717,E2 -7277.717} C_VEL
LIN {X 0,Y 474.978,Z 436.98,A -85,B 0,C 180,E1 -7278.694,E2 -7278.694} C_VEL
LIN {X 0,Y 474.541,Z 445.931,A -85,B 0,C 180,E1 -7279.763,E2 -7279.763} C_VEL
LIN {X 0,Y 474.239,Z 454.689,A -85,B 0,C 180,E1 -7281.048,E2 -7281.048} C_VEL
LIN {X 0,Y 474.034,Z 461.681,A -85,B 0,C 180,E1 -7282.332,E2 -7282.332} C_VEL
LIN {X 0,Y 473.88,Z 467.029,A -85,B 0,C 180,E1 -7283.548,E2 -7283.548} C_VEL
LIN {X 0,Y 473.843,Z 471.68,A -85,B 0,C 180,E1 -7284.894,E2 -7284.894} C_VEL
LIN {X 0,Y 473.788,Z 474,A -85,B 0,C 180,E1 -7285.747,E2 -7285.747} C_VEL
LIN {X 0,Y 473.828,Z 475.888,A -85,B 0,C 180,E1 -7286.599,E2 -7286.599} C_VEL
LIN {X 0,Y 473.865,Z 477.301,A -85,B 0,C 180,E1 -7287.45,E2 -7287.45} C_VEL
LIN {X 0,Y 473.703,Z 478.891,A -85,B 0,C 180,E1 -7289.15,E2 -7289.15} C_VEL
LIN {X 0,Y 473.697,Z 479.095,A -85,B 0,C 180,E1 -7290,E2 -7290} C_VEL
LIN {X 0,Y 473.762,Z 478.226,A -85,B 0,C 180,E1 -7291.7,E2 -7291.7} C_VEL
LIN {X 0,Y 473.868,Z 477.2,A -85,B 0,C 180,E1 -7292.55,E2 -7292.55} C_VEL
LIN {X 0,Y 473.841,Z 475.754,A -85,B 0,C 180,E1 -7293.401,E2 -7293.401} C_VEL
LIN {X 0,Y 473.781,Z 472.724,A -85,B 0,C 180,E1 -7294.68,E2 -7294.68} C_VEL
LIN {X 0,Y 473.863,Z 468.644,A -85,B 0,C 180,E1 -7295.959,E2 -7295.959} C_VEL
LIN {X 0,Y 474.016,Z 462.378,A -85,B 0,C 180,E1 -7297.454,E2 -7297.454} C_VEL
LIN {X 0,Y 474.183,Z 455.542,A -85,B 0,C 180,E1 -7298.738,E2 -7298.738} C_VEL
LIN {X 0,Y 474.454,Z 447.078,A -85,B 0,C 180,E1 -7300.024,E2 -7300.024} C_VEL
LIN {X 0,Y 474.855,Z 438.408,A -85,B 0,C 180,E1 -7301.093,E2 -7301.093} C_VEL
LIN {X 0,Y 475.25,Z 428.275,A -85,B 0,C 180,E1 -7302.116,E2 -7302.116} C_VEL
LIN {X 0,Y 475.671,Z 417.198,A -85,B 0,C 180,E1 -7303.022,E2 -7303.022} C_VEL
LIN {X 0,Y 476.219,Z 405.68,A -85,B 0,C 180,E1 -7303.767,E2 -7303.767} C_VEL
LIN {X 0,Y 476.686,Z 392.557,A -85,B 0,C 180,E1 -7304.406,E2 -7304.406} C_VEL
LIN {X 0,Y 475.277,Z 378.921,A -85,B 0,C 180,E1 -7304.929,E2 -7304.929} C_VEL
LIN {X 0,Y 474.074,Z 369.529,A -85,B 0,C 180,E1 -7305.201,E2 -7305.201} C_VEL
LIN {X 0,Y 474.22,Z 359.673,A -85,B 0,C 180,E1 -7308.133,E2 -7308.133} C_VEL
LIN {X 0,Y 474.456,Z 349.023,A -85,B 0,C 180,E1 -7311.348,E2 -7311.348} C_VEL
LIN {X 0,Y 474.701,Z 338.851,A -85,B 0,C 180,E1 -7314.491,E2 -7314.491} C_VEL
LIN {X 0,Y 475.03,Z 329.713,A -85,B 0,C 180,E1 -7317.415,E2 -7317.415} C_VEL
LIN {X 0,Y 475.51,Z 319.054,A -85,B 0,C 180,E1 -7320.992,E2 -7320.992} C_VEL
LIN {X 0,Y 476.003,Z 310.146,A -85,B 0,C 180,E1 -7324.129,E2 -7324.129} C_VEL
LIN {X 0,Y 476.245,Z 304.65,A -85,B 0,C 180,E1 -7326.178,E2 -7326.178} C_VEL
LIN {X 0,Y 475.344,Z 299.215,A -85,B 0,C 180,E1 -7328.407,E2 -7328.407} C_VEL
LIN {X 0,Y 474.663,Z 295.362,A -85,B 0,C 180,E1 -7330.119,E2 -7330.119} C_VEL
LIN {X 0,Y 474.606,Z 295.37,A -85,B 0,C 180,E1 -7333.481,E2 -7333.481} C_VEL
LIN {X 0,Y 474.606,Z 295.373,A -85,B 0,C 180,E1 -7336.519,E2 -7336.519} C_VEL
LIN {X 0,Y 474.621,Z 295.37,A -85,B 0,C 180,E1 -7339.342,E2 -7339.342} C_VEL
LIN {X 0,Y 474.615,Z 295.368,A -85,B 0,C 180,E1 -7341.704,E2 -7341.704} C_VEL
LIN {X 0,Y 474.629,Z 295.366,A -85,B 0,C 180,E1 -7344.726,E2 -7344.726} C_VEL
LIN {X 0,Y 474.64,Z 295.364,A -85,B 0,C 180,E1 -7347.788,E2 -7347.788} C_VEL
LIN {X 0,Y 474.629,Z 295.366,A -85,B 0,C 180,E1 -7350.885,E2 -7350.885} C_VEL
LIN {X 0,Y 474.666,Z 295.36,A -85,B 0,C 180,E1 -7353.629,E2 -7353.629} C_VEL
LIN {X 0,Y 474.641,Z 295.364,A -85,B 0,C 180,E1 -7356.641,E2 -7356.641} C_VEL
LIN {X 0,Y 474.66,Z 295.361,A -85,B 0,C 180,E1 -7360.09,E2 -7360.09} C_VEL
LIN {X 0,Y 474.644,Z 295.362,A -85,B 0,C 180,E1 -7362.774,E2 -7362.774} C_VEL
LIN {X 0,Y 474.654,Z 295.362,A -85,B 0,C 180,E1 -7365.421,E2 -7365.421} C_VEL
LIN {X 0,Y 474.71,Z 295.357,A -85,B 0,C 180,E1 -7368.038,E2 -7368.038} C_VEL
LIN {X 0,Y 474.715,Z 295.354,A -85,B 0,C 180,E1 -7371.486,E2 -7371.486} C_VEL
LIN {X 0,Y 474.751,Z 295.351,A -85,B 0,C 180,E1 -7374.904,E2 -7374.904} C_VEL
LIN {X 0,Y 474.899,Z 295.331,A -85,B 0,C 180,E1 -7377.455,E2 -7377.455} C_VEL
LIN {X 0,Y 474.918,Z 295.33,A -85,B 0,C 180,E1 -7380,E2 -7380} C_VEL
LIN {X 0,Y 474.9,Z 295.332,A -85,B 0,C 180,E1 -7382.544,E2 -7382.544} C_VEL
LIN {X 0,Y 474.764,Z 295.349,A -85,B 0,C 180,E1 -7385.948,E2 -7385.948} C_VEL
LIN {X 0,Y 474.658,Z 295.363,A -85,B 0,C 180,E1 -7388.515,E2 -7388.515} C_VEL
LIN {X 0,Y 474.376,Z 295.4,A -85,B 0,C 180,E1 -7391.971,E2 -7391.971} C_VEL
LIN {X 0,Y 474.238,Z 298.749,A -85,B 0,C 180,E1 -7395.575,E2 -7395.575} C_VEL
LIN {X 0,Y 474.077,Z 302.082,A -85,B 0,C 180,E1 -7399.035,E2 -7399.035} C_VEL
LIN {X 0,Y 474.045,Z 304.716,A -85,B 0,C 180,E1 -7401.755,E2 -7401.755} C_VEL
LIN {X 0,Y 474.042,Z 305.869,A -85,B 0,C 180,E1 -7402.937,E2 -7402.937} C_VEL
LIN {X 0,Y 477.274,Z 318.479,A -85,B 0,C 180,E1 -7403.45,E2 -7403.45} C_VEL
LIN {X 0,Y 477.04,Z 331.394,A -85,B 0,C 180,E1 -7404.017,E2 -7404.017} C_VEL
LIN {X 0,Y 476.6,Z 343.448,A -85,B 0,C 180,E1 -7404.735,E2 -7404.735} C_VEL
LIN {X 0,Y 476.079,Z 355.008,A -85,B 0,C 180,E1 -7405.619,E2 -7405.619} C_VEL
LIN {X 0,Y 475.683,Z 364.705,A -85,B 0,C 180,E1 -7406.547,E2 -7406.547} C_VEL
LIN {X 0,Y 475.283,Z 373.675,A -85,B 0,C 180,E1 -7407.601,E2 -7407.601} C_VEL
LIN {X 0,Y 474.866,Z 382.801,A -85,B 0,C 180,E1 -7408.93,E2 -7408.93} C_VEL
LIN {X 0,Y 474.51,Z 389.978,A -85,B 0,C 180,E1 -7410.237,E2 -7410.237} C_VEL
LIN {X 0,Y 474.227,Z 396.389,A -85,B 0,C 180,E1 -7411.743,E2 -7411.743} C_VEL
LIN {X 0,Y 474.019,Z 401.282,A -85,B 0,C 180,E1 -7413.269,E2 -7413.269} C_VEL
LIN {X 0,Y 473.935,Z 403.703,A -85,B 0,C 180,E1 -7414.298,E2 -7414.298} C_VEL
LIN {X 0,Y 473.814,Z 405.57,A -85,B 0,C 180,E1 -7415.344,E2 -7415.344} C_VEL
LIN {X 0,Y 473.732,Z 407.075,A -85,B 0,C 180,E1 -7416.763,E2 -7416.763} C_VEL
LIN {X 0,Y 473.728,Z 407.478,A -85,B 0,C 180,E1 -7418.16,E2 -7418.16} C_VEL
LIN {X 0,Y 473.771,Z 406.745,A -85,B 0,C 180,E1 -7419.633,E2 -7419.633} C_VEL
LIN {X 0,Y 473.834,Z 405.267,A -85,B 0,C 180,E1 -7420.848,E2 -7420.848} C_VEL
LIN {X 0,Y 474.022,Z 401.763,A -85,B 0,C 180,E1 -7422.539,E2 -7422.539} C_VEL
LIN {X 0,Y 474.131,Z 398.176,A -85,B 0,C 180,E1 -7423.753,E2 -7423.753} C_VEL
LIN {X 0,Y 474.314,Z 393.625,A -85,B 0,C 180,E1 -7424.958,E2 -7424.958} C_VEL
LIN {X 0,Y 474.493,Z 387.965,A -85,B 0,C 180,E1 -7426.164,E2 -7426.164} C_VEL
LIN {X 0,Y 474.858,Z 380.561,A -85,B 0,C 180,E1 -7427.437,E2 -7427.437} C_VEL
LIN {X 0,Y 475.232,Z 371.91,A -85,B 0,C 180,E1 -7428.64,E2 -7428.64} C_VEL
LIN {X 0,Y 475.675,Z 362.059,A -85,B 0,C 180,E1 -7429.743,E2 -7429.743} C_VEL
LIN {X 0,Y 476.127,Z 351.396,A -85,B 0,C 180,E1 -7430.708,E2 -7430.708} C_VEL
LIN {X 0,Y 476.59,Z 340.449,A -85,B 0,C 180,E1 -7431.498,E2 -7431.498} C_VEL
LIN {X 0,Y 477.001,Z 328.353,A -85,B 0,C 180,E1 -7432.172,E2 -7432.172} C_VEL
LIN {X 0,Y 477.119,Z 318.006,A -85,B 0,C 180,E1 -7432.615,E2 -7432.615} C_VEL
LIN {X 0,Y 473.914,Z 304.647,A -85,B 0,C 180,E1 -7433.152,E2 -7433.152} C_VEL
LIN {X 0,Y 473.919,Z 301.476,A -85,B 0,C 180,E1 -7436.145,E2 -7436.145} C_VEL
LIN {X 0,Y 473.949,Z 298.771,A -85,B 0,C 180,E1 -7438.734,E2 -7438.734} C_VEL
LIN {X 0,Y 473.974,Z 298.172,A -85,B 0,C 180,E1 -7439.297,E2 -7439.297} C_VEL
LIN {X 0,Y 473.352,Z 297.502,A -85,B 0,C 180,E1 -7440.002,E2 -7440.002} C_VEL
LIN {X 0,Y 470.517,Z 296.743,A -85,B 0,C 180,E1 -7441.151,E2 -7441.151} C_VEL
LIN {X 0,Y 468.129,Z 296.418,A -85,B 0,C 180,E1 -7442.079,E2 -7442.079} C_VEL
LIN {X 0,Y 467.153,Z 296.314,A -85,B 0,C 180,E1 -7442.797,E2 -7442.797} C_VEL
LIN {X 0,Y 467.101,Z 296.304,A -85,B 0,C 180,E1 -7443.04,E2 -7443.04} C_VEL
LIN {X 0,Y 467.441,Z 296.26,A -85,B 0,C 180,E1 -7446.049,E2 -7446.049} C_VEL
LIN {X 0,Y 467.586,Z 296.242,A -85,B 0,C 180,E1 -7448.855,E2 -7448.855} C_VEL
LIN {X 0,Y 467.625,Z 296.237,A -85,B 0,C 180,E1 -7451.602,E2 -7451.602} C_VEL
LIN {X 0,Y 467.64,Z 296.233,A -85,B 0,C 180,E1 -7454.305,E2 -7454.305} C_VEL
LIN {X 0,Y 467.657,Z 296.231,A -85,B 0,C 180,E1 -7457.854,E2 -7457.854} C_VEL
LIN {X 0,Y 467.681,Z 296.23,A -85,B 0,C 180,E1 -7461.357,E2 -7461.357} C_VEL
LIN {X 0,Y 467.722,Z 296.224,A -85,B 0,C 180,E1 -7463.962,E2 -7463.962} C_VEL
LIN {X 0,Y 467.86,Z 296.207,A -85,B 0,C 180,E1 -7467.417,E2 -7467.417} C_VEL
LIN {X 0,Y 467.884,Z 296.203,A -85,B 0,C 180,E1 -7470,E2 -7470} C_VEL
LIN {X 0,Y 467.861,Z 296.207,A -85,B 0,C 180,E1 -7472.583,E2 -7472.583} C_VEL
LIN {X 0,Y 467.721,Z 296.226,A -85,B 0,C 180,E1 -7476.038,E2 -7476.038} C_VEL
LIN {X 0,Y 467.681,Z 296.231,A -85,B 0,C 180,E1 -7478.643,E2 -7478.643} C_VEL
LIN {X 0,Y 467.655,Z 296.235,A -85,B 0,C 180,E1 -7482.358,E2 -7482.358} C_VEL
LIN {X 0,Y 467.65,Z 296.232,A -85,B 0,C 180,E1 -7485.885,E2 -7485.885} C_VEL
LIN {X 0,Y 467.622,Z 296.236,A -85,B 0,C 180,E1 -7489.308,E2 -7489.308} C_VEL
LIN {X 0,Y 467.537,Z 296.248,A -85,B 0,C 180,E1 -7492.074,E2 -7492.074} C_VEL
LIN {X 0,Y 467.605,Z 296.238,A -85,B 0,C 180,E1 -7494.887,E2 -7494.887} C_VEL
LIN {X 0,Y 467.621,Z 296.237,A -85,B 0,C 180,E1 -7497.769,E2 -7497.769} C_VEL
LIN {X 0,Y 467.568,Z 296.243,A -85,B 0,C 180,E1 -7501.045,E2 -7501.045} C_VEL
LIN {X 0,Y 467.579,Z 296.243,A -85,B 0,C 180,E1 -7504.24,E2 -7504.24} C_VEL
LIN {X 0,Y 467.55,Z 296.246,A -85,B 0,C 180,E1 -7507.187,E2 -7507.187} C_VEL
LIN {X 0,Y 467.58,Z 296.242,A -85,B 0,C 180,E1 -7510.265,E2 -7510.265} C_VEL
LIN {X 0,Y 467.589,Z 296.241,A -85,B 0,C 180,E1 -7512.567,E2 -7512.567} C_VEL
LIN {X 0,Y 467.568,Z 296.243,A -85,B 0,C 180,E1 -7515.053,E2 -7515.053} C_VEL
LIN {X 0,Y 467.591,Z 296.241,A -85,B 0,C 180,E1 -7517.44,E2 -7517.44} C_VEL
LIN {X 0,Y 467.585,Z 296.241,A -85,B 0,C 180,E1 -7520.856,E2 -7520.856} C_VEL
LIN {X 0,Y 467.562,Z 296.245,A -85,B 0,C 180,E1 -7524.261,E2 -7524.261} C_VEL
LIN {X 0,Y 467.582,Z 296.243,A -85,B 0,C 180,E1 -7527.322,E2 -7527.322} C_VEL
LIN {X 0,Y 467.572,Z 296.242,A -85,B 0,C 180,E1 -7530.668,E2 -7530.668} C_VEL
LIN {X 0,Y 467.591,Z 296.241,A -85,B 0,C 180,E1 -7533.198,E2 -7533.198} C_VEL
LIN {X 0,Y 467.593,Z 296.24,A -85,B 0,C 180,E1 -7536.469,E2 -7536.469} C_VEL
LIN {X 0,Y 467.627,Z 296.238,A -85,B 0,C 180,E1 -7539.777,E2 -7539.777} C_VEL
LIN {X 0,Y 467.602,Z 296.239,A -85,B 0,C 180,E1 -7542.507,E2 -7542.507} C_VEL
LIN {X 0,Y 467.61,Z 296.24,A -85,B 0,C 180,E1 -7545.197,E2 -7545.197} C_VEL
LIN {X 0,Y 467.661,Z 296.233,A -85,B 0,C 180,E1 -7547.855,E2 -7547.855} C_VEL
LIN {X 0,Y 467.674,Z 296.231,A -85,B 0,C 180,E1 -7551.357,E2 -7551.357} C_VEL
LIN {X 0,Y 467.746,Z 296.22,A -85,B 0,C 180,E1 -7553.963,E2 -7553.963} C_VEL
LIN {X 0,Y 467.857,Z 296.207,A -85,B 0,C 180,E1 -7557.417,E2 -7557.417} C_VEL
LIN {X 0,Y 467.886,Z 296.204,A -85,B 0,C 180,E1 -7560,E2 -7560} C_VEL
LIN {X 0,Y 467.853,Z 296.211,A -85,B 0,C 180,E1 -7562.583,E2 -7562.583} C_VEL
LIN {X 0,Y 467.724,Z 296.223,A -85,B 0,C 180,E1 -7566.038,E2 -7566.038} C_VEL
LIN {X 0,Y 467.673,Z 296.231,A -85,B 0,C 180,E1 -7568.643,E2 -7568.643} C_VEL
LIN {X 0,Y 467.661,Z 296.232,A -85,B 0,C 180,E1 -7572.145,E2 -7572.145} C_VEL
LIN {X 0,Y 467.643,Z 296.234,A -85,B 0,C 180,E1 -7575.695,E2 -7575.695} C_VEL
LIN {X 0,Y 467.626,Z 296.237,A -85,B 0,C 180,E1 -7579.308,E2 -7579.308} C_VEL
LIN {X 0,Y 467.539,Z 296.248,A -85,B 0,C 180,E1 -7582.074,E2 -7582.074} C_VEL
LIN {X 0,Y 467.587,Z 296.241,A -85,B 0,C 180,E1 -7584.888,E2 -7584.888} C_VEL
LIN {X 0,Y 467.584,Z 296.242,A -85,B 0,C 180,E1 -7587.772,E2 -7587.772} C_VEL
LIN {X 0,Y 467.572,Z 296.243,A -85,B 0,C 180,E1 -7591.045,E2 -7591.045} C_VEL
LIN {X 0,Y 467.592,Z 296.242,A -85,B 0,C 180,E1 -7594.242,E2 -7594.242} C_VEL
LIN {X 0,Y 467.551,Z 296.244,A -85,B 0,C 180,E1 -7597.186,E2 -7597.186} C_VEL
LIN {X 0,Y 467.575,Z 296.245,A -85,B 0,C 180,E1 -7600.265,E2 -7600.265} C_VEL
LIN {X 0,Y 467.552,Z 296.246,A -85,B 0,C 180,E1 -7603.745,E2 -7603.745} C_VEL
LIN {X 0,Y 467.552,Z 296.244,A -85,B 0,C 180,E1 -7606.255,E2 -7606.255} C_VEL
LIN {X 0,Y 467.597,Z 296.263,A -85,B 0,C 180,E1 -7609.666,E2 -7609.666} C_VEL
LIN {X 0,Y 469.239,Z 305.144,A -85,B 0,C 180,E1 -7613.194,E2 -7613.194} C_VEL
LIN {X 0,Y 469.386,Z 309.491,A -85,B 0,C 180,E1 -7614.798,E2 -7614.798} C_VEL
LIN {X 0,Y 468.886,Z 318.145,A -85,B 0,C 180,E1 -7617.852,E2 -7617.852} C_VEL
LIN {X 0,Y 468.359,Z 328.291,A -85,B 0,C 180,E1 -7621.303,E2 -7621.303} C_VEL
LIN {X 0,Y 467.919,Z 338.661,A -85,B 0,C 180,E1 -7624.717,E2 -7624.717} C_VEL
LIN {X 0,Y 467.511,Z 348.67,A -85,B 0,C 180,E1 -7627.925,E2 -7627.925} C_VEL
LIN {X 0,Y 467.282,Z 359.628,A -85,B 0,C 180,E1 -7631.358,E2 -7631.358} C_VEL
LIN {X 0,Y 467.036,Z 370.099,A -85,B 0,C 180,E1 -7634.585,E2 -7634.585} C_VEL
LIN {X 0,Y 468.978,Z 385.419,A -85,B 0,C 180,E1 -7635.074,E2 -7635.074} C_VEL
LIN {X 0,Y 469.756,Z 393.886,A -85,B 0,C 180,E1 -7635.432,E2 -7635.432} C_VEL
LIN {X 0,Y 469.313,Z 405.742,A -85,B 0,C 180,E1 -7636.026,E2 -7636.026} C_VEL
LIN {X 0,Y 468.79,Z 417.256,A -85,B 0,C 180,E1 -7636.784,E2 -7636.784} C_VEL
LIN {X 0,Y 468.264,Z 428.527,A -85,B 0,C 180,E1 -7637.723,E2 -7637.723} C_VEL
LIN {X 0,Y 467.873,Z 438.376,A -85,B 0,C 180,E1 -7638.739,E2 -7638.739} C_VEL
LIN {X 0,Y 467.434,Z 446.996,A -85,B 0,C 180,E1 -7639.824,E2 -7639.824} C_VEL
LIN {X 0,Y 467.12,Z 455.387,A -85,B 0,C 180,E1 -7641.129,E2 -7641.129} C_VEL
LIN {X 0,Y 466.926,Z 462.156,A -85,B 0,C 180,E1 -7642.432,E2 -7642.432} C_VEL
LIN {X 0,Y 466.774,Z 468.361,A -85,B 0,C 180,E1 -7643.95,E2 -7643.95} C_VEL
LIN {X 0,Y 466.702,Z 472.384,A -85,B 0,C 180,E1 -7645.249,E2 -7645.249} C_VEL
LIN {X 0,Y 466.757,Z 475.355,A -85,B 0,C 180,E1 -7646.547,E2 -7646.547} C_VEL
LIN {X 0,Y 466.775,Z 476.768,A -85,B 0,C 180,E1 -7647.411,E2 -7647.411} C_VEL
LIN {X 0,Y 466.698,Z 477.761,A -85,B 0,C 180,E1 -7648.274,E2 -7648.274} C_VEL
LIN {X 0,Y 466.624,Z 478.561,A -85,B 0,C 180,E1 -7650,E2 -7650} C_VEL
LIN {X 0,Y 466.634,Z 478.324,A -85,B 0,C 180,E1 -7650.863,E2 -7650.863} C_VEL
LIN {X 0,Y 466.792,Z 476.657,A -85,B 0,C 180,E1 -7652.589,E2 -7652.589} C_VEL
LIN {X 0,Y 466.77,Z 475.208,A -85,B 0,C 180,E1 -7653.453,E2 -7653.453} C_VEL
LIN {X 0,Y 466.707,Z 472.171,A -85,B 0,C 180,E1 -7654.751,E2 -7654.751} C_VEL
LIN {X 0,Y 466.775,Z 468.082,A -85,B 0,C 180,E1 -7656.05,E2 -7656.05} C_VEL
LIN {X 0,Y 466.926,Z 461.807,A -85,B 0,C 180,E1 -7657.568,E2 -7657.568} C_VEL
LIN {X 0,Y 467.112,Z 454.968,A -85,B 0,C 180,E1 -7658.872,E2 -7658.872} C_VEL
LIN {X 0,Y 467.412,Z 446.503,A -85,B 0,C 180,E1 -7660.176,E2 -7660.176} C_VEL
LIN {X 0,Y 467.863,Z 437.833,A -85,B 0,C 180,E1 -7661.261,E2 -7661.261} C_VEL
LIN {X 0,Y 468.26,Z 427.937,A -85,B 0,C 180,E1 -7662.277,E2 -7662.277} C_VEL
LIN {X 0,Y 468.71,Z 416.619,A -85,B 0,C 180,E1 -7663.219,E2 -7663.219} C_VEL
LIN {X 0,Y 469.291,Z 405.121,A -85,B 0,C 180,E1 -7663.974,E2 -7663.974} C_VEL
LIN {X 0,Y 469.783,Z 392.041,A -85,B 0,C 180,E1 -7664.623,E2 -7664.623} C_VEL
LIN {X 0,Y 468.326,Z 379.214,A -85,B 0,C 180,E1 -7665.134,E2 -7665.134} C_VEL
LIN {X 0,Y 466.997,Z 368.988,A -85,B 0,C 180,E1 -7665.432,E2 -7665.432} C_VEL
LIN {X 0,Y 467.18,Z 358.52,A -85,B 0,C 180,E1 -7668.605,E2 -7668.605} C_VEL
LIN {X 0,Y 467.405,Z 348.757,A -85,B 0,C 180,E1 -7671.616,E2 -7671.616} C_VEL
LIN {X 0,Y 467.688,Z 338.466,A -85,B 0,C 180,E1 -7674.883,E2 -7674.883} C_VEL
LIN {X 0,Y 468.037,Z 329.706,A -85,B 0,C 180,E1 -7677.742,E2 -7677.742} C_VEL
LIN {X 0,Y 468.554,Z 319.486,A -85,B 0,C 180,E1 -7681.244,E2 -7681.244} C_VEL
LIN {X 0,Y 469.105,Z 310.428,A -85,B 0,C 180,E1 -7684.513,E2 -7684.513} C_VEL
LIN {X 0,Y 469.298,Z 306.437,A -85,B 0,C 180,E1 -7686.033,E2 -7686.033} C_VEL
LIN {X 0,Y 468.624,Z 301.799,A -85,B 0,C 180,E1 -7687.944,E2 -7687.944} C_VEL
LIN {X 0,Y 467.599,Z 296.241,A -85,B 0,C 180,E1 -7690.475,E2 -7690.475} C_VEL
LIN {X 0,Y 467.56,Z 296.249,A -85,B 0,C 180,E1 -7693.744,E2 -7693.744} C_VEL
LIN {X 0,Y 467.56,Z 296.251,A -85,B 0,C 180,E1 -7696.256,E2 -7696.256} C_VEL
LIN {X 0,Y 467.582,Z 296.245,A -85,B 0,C 180,E1 -7698.723,E2 -7698.723} C_VEL
LIN {X 0,Y 467.57,Z 296.246,A -85,B 0,C 180,E1 -7701.956,E2 -7701.956} C_VEL
LIN {X 0,Y 467.569,Z 296.244,A -85,B 0,C 180,E1 -7705.168,E2 -7705.168} C_VEL
LIN {X 0,Y 467.588,Z 296.243,A -85,B 0,C 180,E1 -7708.26,E2 -7708.26} C_VEL
LIN {X 0,Y 467.582,Z 296.243,A -85,B 0,C 180,E1 -7711.251,E2 -7711.251} C_VEL
LIN {X 0,Y 467.622,Z 296.239,A -85,B 0,C 180,E1 -7713.2,E2 -7713.2} C_VEL
LIN {X 0,Y 467.598,Z 296.241,A -85,B 0,C 180,E1 -7716.468,E2 -7716.468} C_VEL
LIN {X 0,Y 467.628,Z 296.237,A -85,B 0,C 180,E1 -7719.777,E2 -7719.777} C_VEL
LIN {X 0,Y 467.604,Z 296.239,A -85,B 0,C 180,E1 -7722.506,E2 -7722.506} C_VEL
LIN {X 0,Y 467.612,Z 296.24,A -85,B 0,C 180,E1 -7725.196,E2 -7725.196} C_VEL
LIN {X 0,Y 467.662,Z 296.233,A -85,B 0,C 180,E1 -7727.855,E2 -7727.855} C_VEL
LIN {X 0,Y 467.673,Z 296.231,A -85,B 0,C 180,E1 -7731.357,E2 -7731.357} C_VEL
LIN {X 0,Y 467.724,Z 296.225,A -85,B 0,C 180,E1 -7733.962,E2 -7733.962} C_VEL
LIN {X 0,Y 467.864,Z 296.208,A -85,B 0,C 180,E1 -7737.417,E2 -7737.417} C_VEL
LIN {X 0,Y 467.888,Z 296.206,A -85,B 0,C 180,E1 -7740,E2 -7740} C_VEL
LIN {X 0,Y 467.865,Z 296.208,A -85,B 0,C 180,E1 -7742.583,E2 -7742.583} C_VEL
LIN {X 0,Y 467.727,Z 296.226,A -85,B 0,C 180,E1 -7746.037,E2 -7746.037} C_VEL
LIN {X 0,Y 467.619,Z 296.24,A -85,B 0,C 180,E1 -7748.644,E2 -7748.644} C_VEL
LIN {X 0,Y 467.337,Z 296.383,A -85,B 0,C 180,E1 -7752.176,E2 -7752.176} C_VEL
LIN {X 0,Y 467.178,Z 299.738,A -85,B 0,C 180,E1 -7755.711,E2 -7755.711} C_VEL
LIN {X 0,Y 467.065,Z 302.46,A -85,B 0,C 180,E1 -7758.562,E2 -7758.562} C_VEL
LIN {X 0,Y 467.022,Z 304.98,A -85,B 0,C 180,E1 -7761.172,E2 -7761.172} C_VEL
LIN {X 0,Y 467.013,Z 306.539,A -85,B 0,C 180,E1 -7762.712,E2 -7762.712} C_VEL
LIN {X 0,Y 470.453,Z 319.8,A -85,B 0,C 180,E1 -7763.255,E2 -7763.255} C_VEL
LIN {X 0,Y 470.211,Z 331.917,A -85,B 0,C 180,E1 -7763.801,E2 -7763.801} C_VEL
LIN {X 0,Y 469.771,Z 343.352,A -85,B 0,C 180,E1 -7764.485,E2 -7764.485} C_VEL
LIN {X 0,Y 469.295,Z 353.651,A -85,B 0,C 180,E1 -7765.265,E2 -7765.265} C_VEL
LIN {X 0,Y 468.792,Z 364.529,A -85,B 0,C 180,E1 -7766.294,E2 -7766.294} C_VEL
LIN {X 0,Y 468.386,Z 372.646,A -85,B 0,C 180,E1 -7767.235,E2 -7767.235} C_VEL
LIN {X 0,Y 467.987,Z 381.43,A -85,B 0,C 180,E1 -7768.477,E2 -7768.477} C_VEL
LIN {X 0,Y 467.614,Z 388.598,A -85,B 0,C 180,E1 -7769.734,E2 -7769.734} C_VEL
LIN {X 0,Y 467.342,Z 394.421,A -85,B 0,C 180,E1 -7770.998,E2 -7770.998} C_VEL
